FUNCTION_BLOCK "STD_DUMPFlowMonitor"	// FB 1804
TITLE = DUMP-Scale test productflow
//COPYRIGHT:    (C) 2004  BUHLER AG, CH-9240 UZWIL, SWITZERLAND
//
//PRODUCT:      STD_MU664
//
//TITLE:        Test product flow dump scale
//
//              Überprüfen des Produktflusses mit Schüttwaage
//
//
//--------------------------------------------------------------------------------
//
//IDENT:         AUTHOR:             DEPT:                             DATE:
//
//STD_FB1804.3.0 Ph. Engler          MU92                              24-May-2005
//               - InReadyForScaleEmptying
//STD_FB1804.2.0 Ph. Engler          MU92                              11-May-2005
//               - Timer type changed to FB1706
//               - S5Timer 40 changed with an Timer-FB1706
//STD_FB1804.1.0 E.Hanselmann        MU662                             26-Mar-2003
//               1st Release
//
//--------------------------------------------------------------------------------
//
//PURPOSE: 
//
//MANUAL : 
//
//RESTRICTIONS: 
//
//--------------------------------------------------------------------------------
//
AUTHOR : PE
FAMILY : STD
VERSION : 3.0
VAR_INPUT
  InFuncCode : INT ;	//0=nothing,1=DUMP, 2=not used,3=not used,
  InInit : BOOL ;	//(S-DB.ToASW.CmdNewBatch)
  InScaleWeight : DINT ;	//Actual scale weight (#xxx.xxx.OutScaleWeight)
  InJobWeight : DINT ;	//[not used] Actual job weight   (#xxx.xxx.OutJobWeight)
  InFlowrate : DINT ;	//[not used] Actual scale flowrate (#xxx.xxx.OutFlowrate)
  InDumpWeight : INT ;	//Adjusted dump weight scale (#xxx.xxx.DUMP.InDumpWeight)
  InStepScale : INT ;	//Actual scale step  (#xxx.xxx.OutLcStep)
  InFlowMeasureTime : INT ;	//Interval to meassuring product flow (seconds/minutes)
  InMinFlowWeightPerTime : DINT ;	//Minimal weight per messure cycle "NoProductFlow"
  InDelaySeqStopTime : INT ;	//Delay SequenceStop after "NoProductFlow" (seconds/minutes)
  InSectionStarted : BOOL ;	//(S-DB.PcRead.State.StStarted)
  InSectionFeeding : BOOL ;	//(S-DB.PcRead.State.StFeeding)
  InGroupLoaded : BOOL ;	//[not used] (#Gr.OutLoaded)
  InReadyForScaleEmptying : BOOL ;	//The section is ready to monitor the scale for no material flow.
END_VAR
VAR
  FlowMeasureTimer : FB 1706;
  DelaySeqStopTimer : FB 1706;
  WaitForProductDelay : FB 1706;
  OutScaleProductFlowOn : BOOL ;	//Used for "  "
  OutScaleLoaded : BOOL ;	//Used for "  "
  OutReadyRestEmptying : BOOL ;	//Used for cmd "RestEmptying" (#xxx.Ma.InOutEmptyingHopperScale)
  OutProductFlowEnd : BOOL ;	//Used for "SequenzeStop" (S-DB.ToSSW.Func.CmdSequenzStop)
  OutActProductFlowPerTime : DINT ;	//Actual product flow
  ProductWeightOld : DINT ;	//Weight by last cycle
  ProductWeightNew : DINT ;	//Weight by actual cycle
  JobWeightOld : DINT ;	//Weight by last cycle
END_VAR
BEGIN
NETWORK
TITLE = General
      A(;
      L     #InFuncCode;
      L     0;	//Timer type "nothing"
      <=I;
      );
      O;
      A(;
      L     #InFuncCode;
      L     2;	//Timer type "not used"
      >=I;
      );
      BEC;
NETWORK
TITLE = Flow Measure Time Intervall
      NOP   0;
//-Waiting for product---
      L     #InStepScale;
      L     8;	//step wait product
      ==I;
      AN    #FlowMeasureTimer.Q;
      =     #WaitForProductDelay.IN;
// 
      CALL  #WaitForProductDelay (
           TON                      := TRUE,
           ParRestart               := FALSE,
           ParRecalc                := FALSE,
           PT                       := 20);
      L     #InStepScale;
      L     2;
      ==I;
      O     #WaitForProductDelay.Q;
      AN    #FlowMeasureTimer.Q;
// 
//-Intervall for measureing---
      =     #FlowMeasureTimer.IN;
      L     #InFlowMeasureTime;	//step dosing
      T     #FlowMeasureTimer.PT;
//Target Time
      CALL  #FlowMeasureTimer (
           TON                      := TRUE,
           ParRestart               := FALSE,
           ParRecalc                := FALSE);
//Timer
NETWORK
TITLE = Product Flow
      NOP   0;
//Meassure Flow
      L     L#0;
      A     #FlowMeasureTimer.Q;
      JCN   PF04;
      A(;
      L     #InScaleWeight;
      L     L#0;
      <D;
      );
      JC    PF01;
      TAK;
PF01: T     #ProductWeightNew;
// 
      A(;
      L     #ProductWeightNew;
      L     #ProductWeightOld;
      >=D;
      );
      JC    PF02;
      A(;
      L     #ProductWeightNew;
      L     #ProductWeightOld;
      <D;
      );
      JU    PF03;
PF02: L     #ProductWeightNew;
      L     #ProductWeightOld;
      -D;
      JU    PF04;
PF03: L     #InDumpWeight;
      ITD;
      L     1000;	//kg to gr
      *D;
      L     #ProductWeightOld;
      -D;
      L     #ProductWeightNew;
      +D;
      JU    PF04;
PF04: T     #OutActProductFlowPerTime;
      L     #ProductWeightNew;
      T     #ProductWeightOld;
// 
      A(;
      L     #OutActProductFlowPerTime;
      L     #InMinFlowWeightPerTime;
      >=D;
      );
      O(;
      L     #InJobWeight;
      L     #JobWeightOld;
      >D;
      );
      A(;
      O     #InSectionStarted;
      O     #InSectionFeeding;
      );
      S     #OutScaleProductFlowOn;
      S     #OutScaleLoaded;
      A(;
      L     #OutActProductFlowPerTime;
      L     #InMinFlowWeightPerTime;
      <D;
      );
      A     #FlowMeasureTimer.Q;
      R     #OutScaleProductFlowOn;
      L     #InJobWeight;
      T     #JobWeightOld;
// 
//Initialize
      A     #InInit;
      JCN   PF06;
      SET;
      R     #OutScaleProductFlowOn;
      R     #OutScaleLoaded;
      L     L#0;
      T     #ProductWeightNew;
      T     #ProductWeightOld;
      T     #OutActProductFlowPerTime;
PF06: NOP   0;
NETWORK
TITLE = Ready Rest Emptying
      A(;
      O     #InSectionStarted;
      O     #InSectionFeeding;
      );
      A     #FlowMeasureTimer.Q;
      A     #OutScaleLoaded;
      AN    #OutScaleProductFlowOn;
      S     #OutReadyRestEmptying;
//Initialize
      A     #InInit;
      O;
      A     #OutScaleLoaded;
      A     #OutScaleProductFlowOn;
      AN    #InReadyForScaleEmptying;
      R     #OutReadyRestEmptying;
NETWORK
TITLE = Delay SequenzeStop Time
      NOP   0;
//Start
      L     #InDelaySeqStopTime;
      L     0;
      >I;
      A     #InSectionFeeding;
      A     #OutScaleLoaded;
      AN    #OutScaleProductFlowOn;
      =     #DelaySeqStopTimer.IN;
//Target Time
      L     #InDelaySeqStopTime;
      T     #DelaySeqStopTimer.PT;
//Timer
      CALL  #DelaySeqStopTimer (
           TON                      := TRUE,
           ParRestart               := FALSE,
           ParRecalc                := FALSE);
NETWORK
TITLE = Product Flow End
      A     #DelaySeqStopTimer.Q;
      =     #OutProductFlowEnd;
NETWORK
TITLE = End of block
      BE;
END_FUNCTION_BLOCK

FUNCTION_BLOCK "STD_DUMPPulse"	// FB 1805
TITLE = Handling of Scales with Dump Impuls
//COPYRIGHT:    (C) 2004  BUHLER AG, CH-9240 UZWIL, SWITZERLAND
//
//PRODUCT:      STD
//
//TITLE:        Handling of Scales with Dump Impuls
//
//              Schüttimpulsauswertung
//                
// 
//--------------------------------------------------------------------------------
// 
//IDENT:            AUTHOR:             DEPT:                          DATE:
// 
//STD_FB1805.2.0    Ph. Engler          MU664                          03-Jun-2004
//                  Integration to GP-BIB; New functionality
//P02_FB1805.1.1    M.Miotto            MU662                          11-May-2004
//                  Init if no dump after a predefined time >> from 180 decr. 60
//P02_FB1805.1.0    P.Müller            MU662                          30-Apr-2004
//                  1st Release
// 
//--------------------------------------------------------------------------------
// 
//PURPOSE: 
// 
//MANUAL : 
// 
//RESTRICTIONS: 
// 
//--------------------------------------------------------------------------------
//
AUTHOR : PE
FAMILY : STD
VERSION : 2.0
VAR_INPUT
  FunctionCode : INT ;
  InFeeding : BOOL ;
  CmdNewJob : BOOL ;
  CmdNewValue : BOOL ;
  ScalePulse : BOOL ;
  ScalePulseWeight : DINT ;
  TargetFlowrate : INT ;
END_VAR
VAR_OUTPUT
  InfScaleDumpRelease : BOOL ;
END_VAR
VAR_IN_OUT
  ScaleJobWeight : DINT ;
  ScaleNonErasableWeight : DINT ;
  ScaleActualFlowrate : DINT ;
END_VAR
VAR
  TimeCounter : DINT ;
  ScaleDumpTimer : INT ;
  DumpMonitoringTimer : INT ;
  EdgeScalePulse : BOOL ;
  PulseScalePulse : BOOL ;
  ScaleFeeding : BOOL ;
  staFirstDumpDone : BOOL ;
  EdgeInFeeding : BOOL ;
  PulseInFeeding : BOOL ;
  InfDumpMonitoringElapsed : BOOL ;
  staScaleNotDumping : BOOL ;
  staNewFlowrate : BOOL ;
  AverageTime : INT ;
  StartTime : INT ;
  ActDumpIntervallTime : ARRAY  [1 .. 3 ] OF INT ;
END_VAR
VAR_TEMP
  tmpMaxPulsesPerHour : REAL ;
  tmpPulseTime : DINT ;
  tmpNumberOfTimeValues : INT ;
  tmpInputIntervallTime : INT ;
END_VAR
BEGIN
NETWORK
TITLE = Function 1: Calculation of Target Flowrate
      L     #FunctionCode;
      L     1;
      <>I;
      JC    F001;
// 
//-Calculation of Pulse per Hour---
      L     #TargetFlowrate;
      ITD;
      DTR;
      L     #ScalePulseWeight;
      DTR;
      /R;
      T     #tmpMaxPulsesPerHour;
// 
//-Calculation of Pulse Pause---
      L     3.600000e+03;
      L     #tmpMaxPulsesPerHour;
      /R;
      RND;
      T     #tmpPulseTime;
// 
//-Release Scale Dump---
      A     "SYS_Scan0_Tick1s";
      JCN   NE10;
      L     #TimeCounter;
      L     L#1;
      +D;
      T     #TimeCounter;
NE10: L     #tmpPulseTime;
      L     #TimeCounter;
      <=D;
      =     #InfScaleDumpRelease;
      JCN   NE11;
      L     L#0;
      T     #TimeCounter;
NE11: NOP   0;
// 
      BEU;
F001: NOP   0;
NETWORK
TITLE = Function 2: Calculation of Scale Values
//Scale Values:
//- Job Weight
//- Non Erasable Weight
//- Flowrate
      L     #FunctionCode;
      L     2;
      <>I;
      JC    F002;
// 
//-Weight calculatione---
      A     #PulseScalePulse;
      JCN   NE22;
      L     #ScalePulseWeight;
      L     #ScaleJobWeight;
      +D;
      T     #ScaleJobWeight;
// 
      L     #ScalePulseWeight;
      L     #ScaleNonErasableWeight;
      +D;
      T     #ScaleNonErasableWeight;
NE22: NOP   0;
// 
//-Dump intervall time measuring---
      A     #InFeeding;
      A     "SYS_Scan0_Tick1s";
      JCN   NE23;
      L     L#1;
      L     #ScaleDumpTimer;
      +D;
      T     #ScaleDumpTimer;
NE23: NOP   0;
// 
//-CmdNewValue---
      A     #CmdNewValue;
      O     #CmdNewJob;
      S     #staNewFlowrate;
// 
//-Dump monitoring---
      L     0;
//      U     #InFeeding
//      SPBN  DM02
      A     "SYS_Scan0_Tick1s";
      JCN   DM01;
      L     L#1;
      L     #DumpMonitoringTimer;
      +D;
      T     #DumpMonitoringTimer;
DM01: NOP   0;
// 
      AN    #staScaleNotDumping;
      O     #staNewFlowrate;
      JCN   DM03;
      L     #AverageTime;
      L     2;
      /I;
      L     #AverageTime;
      +I;
      JU    DM04;
DM03: L     #AverageTime;
      L     2;
      /I;
DM04: L     #DumpMonitoringTimer;
      <=I;
      A(;
      TAK;
      L     0;
      <>I;
      );
      =     #InfDumpMonitoringElapsed;
      S     #staScaleNotDumping;
// 
//-Number of valid DumpIntervall times---
      L     0;
      T     #tmpNumberOfTimeValues;
      L     #ActDumpIntervallTime[1];
      <>I;
      JCN   AcD1;
      L     1;
      L     #tmpNumberOfTimeValues;
      +I;
      T     #tmpNumberOfTimeValues;
AcD1: L     0;
      L     #ActDumpIntervallTime[2];
      <>I;
      JCN   AcD2;
      L     1;
      L     #tmpNumberOfTimeValues;
      +I;
      T     #tmpNumberOfTimeValues;
AcD2: L     0;
      L     #ActDumpIntervallTime[3];
      <>I;
      JCN   AcD3;
      L     1;
      L     #tmpNumberOfTimeValues;
      +I;
      T     #tmpNumberOfTimeValues;
AcD3: NOP   0;
// 
//-InFeeding---
      A     #InFeeding;
      FP    #EdgeInFeeding;
      =     #PulseInFeeding;
// 
//-Scale dump pulse---
      A     #ScalePulse;
      FP    #EdgeScalePulse;
      =     #PulseScalePulse;
      R     #staScaleNotDumping;
      R     #staNewFlowrate;
// 
//-Save intervall times---
      L     0;
      A     #InfDumpMonitoringElapsed;
      JC    IT01;
      L     #StartTime;
      AN    #staFirstDumpDone;
      JC    IT01;
      L     #ScaleDumpTimer;
IT01: T     #tmpInputIntervallTime;
      A     #PulseScalePulse;
      O     #InfDumpMonitoringElapsed;
      JCN   SI02;
      L     #ActDumpIntervallTime[2];
      T     #ActDumpIntervallTime[3];
      L     #ActDumpIntervallTime[1];
      T     #ActDumpIntervallTime[2];
      L     #tmpInputIntervallTime;
      T     #ActDumpIntervallTime[1];
      L     L#0;
      T     #DumpMonitoringTimer;
      A     #PulseScalePulse;
      JCN   SI02;
      T     #ScaleDumpTimer;
SI02: NOP   0;
// 
//-First dump after inFeeding on---
      A     #PulseScalePulse;
      AN    #staFirstDumpDone;
      S     #staFirstDumpDone;
      AN    #InFeeding;
      R     #staFirstDumpDone;
// 
//-New job/ job change---
      A     #CmdNewJob;
      JCN   NJ01;
//      L     #ActDumpIntervallTime[1]
//      T     #ActDumpIntervallTime[2]
//      L     0
//      T     #ActDumpIntervallTime[1]
//      T     #ActDumpIntervallTime[3]
// 
      L     L#0;
      T     #ScaleJobWeight;
NJ01: NOP   0;
// 
//-Time average---
      L     #ActDumpIntervallTime[1];
      L     #ActDumpIntervallTime[2];
      +I;
      L     #ActDumpIntervallTime[3];
      +I;
      L     #tmpNumberOfTimeValues;
      /I;
      T     #AverageTime;
// 
//-Start time---
      L     0;
      L     #AverageTime;
      <>I;
      JCN   ST01;
      L     #AverageTime;
      T     #StartTime;
ST01: NOP   0;
// 
//-Flowrate---
      L     0;
      A     #InFeeding;
      JCN   FL01;
      L     #ScalePulseWeight;
      L     L#3600;
      *D;
      L     #AverageTime;
      /D;
FL01: T     #ScaleActualFlowrate;
// 
//-Scale feeding---
      L     #ScaleActualFlowrate;
      L     0;
      >I;
      A     #InFeeding;
      =     #ScaleFeeding;
// 
      SET;
      R     #CmdNewValue;
      R     #CmdNewJob;
// 
      BEU;
F002: NOP   0;
NETWORK
TITLE = End of block
      BE;
END_FUNCTION_BLOCK

// FC 6: know-how protected block, not included

// FC 8: know-how protected block, not included

FUNCTION "SYS_DPDiag1" : VOID	// FC 76
TITLE = DP-additional Diag
//COPYRIGHT:     (C) 2001 BY  BUEHLER LTD. 
//                            CH-9240 UZWIL  SWITZERLAND
//
//PRODUCT:       DP-Diagnosis
//
//TITLE:         DP-additional Diag
//
//-------------------------------------------------------------------------
//
//IDENT:        AUTOR:              DEPT:                         DATE:
//
//FC76.2.0      Ph. Engler          MU664                        14-Dec-2004
//              Wago 750-333: Corrections and adaption to WinCC
//FC76.1B       K. Tischer          CT3                          20-Feb-2003
//              new buskoppler Wago 750-333 added
//FC76.1A       K. Tischer          CT3                          28-MAY-2001
//              1st Release
//
//-------------------------------------------------------------------------
//
//PURPOSE:  - each mastersystem is a separate Network
//              - initial same Bit
//              - Call DP-Diagnostic (orig. Siemens) 
//              - Call additional Diagnostic for not Siemens Slaves
//              - reset same parameters
//
//RESTRICTIONS:   NEEDS SIEMENS FB76 (original FB125)
//                NEEDS FC75 Main Diagnostic
//
//
//-------------------------------------------------------------------------
//
//
AUTHOR : PE
FAMILY : DP
NAME : DPDiag1
VERSION : 2.0
VAR_TEMP
  Sum_Slave_Diag_Int : BYTE ;	//summary Slave Diagnosen
  ErrorNo : BYTE ;	//TiK
  ByteStart : INT ;	//TiK
  Diag_Lentgh : BYTE ;	//TiK
  Adr : DINT ;	//adress1
  Adr2 : DINT ;	//Adress 2
END_VAR
BEGIN
NETWORK
TITLE = check is diagtic present
      AN    DBX 932.3;	// additional diagnostic data present
      BEC;
NETWORK
TITLE = WAxx Wago (B750) 
//additianal Diagnisis for Wago Slaves Type (B750)
//
// - check result from SIEMENS FB76 => error type = device diagnosis
// - check result from SIEMENS FB76 => slave ident = B750
//
      NOP   0;
// error type = device diagnosis
      A(;
      L     DBB 11;	// error typ
      L     5;	// check device diagnostic
      ==I;
      );
// slave ident = B750
      A(;
      L     DBW 8;	// slave ident
      L     W#16#B750;	// B750 = Wago
      ==I;
      );
      JCN   WA00;	// jump end
// Init wago standard
      L     8;	// standard length of wago diagnostic data
      T     #Diag_Lentgh;
      L     DBB 1398;	// old error no (stored)
      T     #ErrorNo;	// error no
// calc summary DiagData
      L     DBB 938;	// norm diag data byte 6 (length)
      +     -2;	// 2 byte length info
      L     #Diag_Lentgh;	// Wago standard length =8
      /I;
      T     #Sum_Slave_Diag_Int;	// summary diag data
// Diag counter intialisieren
      A     DBX 2.3;	// single step error
      JCN   WA07;
// Diag counter inkrementieren
      L     #ErrorNo;	// actual diagnostic data no
      +     1;	// inkrement 1
      T     #ErrorNo;	// actual diagnostic data no
// Diag conter upper and lower limit
WA07: A(;
      L     #ErrorNo;
      L     #Sum_Slave_Diag_Int;	// upper limit 
      >I;
      );
      O(;
      L     #ErrorNo;
      L     1;	// lower limit
      <I;
      );
      JCN   WA06;
      L     1;	// set count diag =1
      T     #ErrorNo;	// out of range
WA06: NOP   0;
// write diagnostic to siemens DB
      L     #ErrorNo;
      T     DBB 10;	// => error number
      T     DBB 1398;	// => reserve byte siemens to store old error number
// calc start byte
      L     #ErrorNo;	// actual diagnostic data no
      L     #Diag_Lentgh;	// length diagnostic data
      *D;	// offset to start byte
      L     932;	// start byte diagnostic data
      +D;
      T     #ByteStart;	// => byte src diagnostic data
// ==check for Profibus or Klemmbus Diagnosis (first byte diagnostic data=0)===================      
      L     0;	// byte no
      L     #ByteStart;	// byte no start actual data
      +D;
      SLD   3;	// convert to bit value
      T     #Adr;	// store bit value
      L     DBB [#Adr];	// first byte diagnostic data
      L     0;
      ==I;
      JC    WA02;	//>>jump to check Klembus diagnosis >>>>>>>>>>>>>>>>>>>
// Modul / Kanal Diagnose ============================
      L     DBB [#Adr];	// first byte diagnostic data
      T     DBB 12;	// => modul no
      L     1;	// byte no
      L     #ByteStart;	// byte no start actual data
      +D;
      SLD   3;	// convert to bit value
      T     #Adr;	// store bit value
      L     DBB [#Adr];
      T     DBB 14;	// => cannel no
// Error analyse
      L     4;	// byte no
      L     #ByteStart;	// byte no start actual data
      +D;
      SLD   3;	// convert to bit value
      T     #Adr;	// store bit value
// == check Lower limit violated ======
      L     DBB [#Adr];
      L     2#100000001;	// compare bit 0 set
      AW;
      L     0;
      JCN   WA05;	// >> jump to check overrange >>>>>>>>>>>>>>>>>>>>>>>>>
      L     8;	//  8=Lower limit violated
      JU    WA03;	// >> jump to => canal error code >>>>>>>>>>>>>>>>>>>>>
// == check Upper limit violated ======
WA05: L     DBB [#Adr];
      L     2#100000010;	// compare bit 1 set
      AW;
      JCN   WA04;	// >> jump to other fault
      L     7;	// 7=Upper limit violated
      JU    WA03;	// >> jump to => canal error code >>>>>>>>>>>>>>>>>>>>>
WA04: L     DBB [#Adr];
      L     2#101000000;	// compare bit 6 set
      AW;
      JCN   WA03;	// >> jump to => canal error code >>>>>>>>>>>>>>>>>>>>>
      L     9;	// 9= Fault (e.g. encoder supply, load voltage at the output...;
WA03: T     DBW 16;	// => canal error code
      L     3;	// 3= channel error
      T     DBB 11;	// => error type
      JU    WA00;	// jump end
WA02: NOP   0;	// << check Klemmbus diagnosis <<<<<<<<<<<<<<<<<<<<<<<<<
      L     1;	// byte no
      L     #ByteStart;	// byte no start actual data
      +D;
      SLD   3;	// convert to bit value
      T     #Adr;	// store bit value
      L     DBB [#Adr];
      L     0;
      ==I;
      JC    WA01;	//>>jump to Klemmbus diagnosis >>>>>>>>>>>>>>>>>>>>>>>>>
// Profibus Diagnosis =================================
      L     4;	// byte no
      L     #ByteStart;	// byte no start actual data
      +D;
      SLD   3;	// convert to bit value
      T     #Adr;	// store bit value
      L     DBB [#Adr];
      L     100;	// 100=not enough configuration data;200=error in 1st configuration byte;300=non-supported module at position N
      *I;
      T     DBB 13;	// => modul state
      L     2;	// 2=Modul Diagnosis
      T     DBB 11;	// => error type
      JU    WA00;	// >> jump end >>>>>>>>>>>>>>>>>>>>>>>>>>>>>>>>>>>>>>>>>>>
// << Klemmenbus Diagnosis <<<<<<<<<<<<<<<<<<<<<<<<<<<<<<<
WA01: NOP   0;
// prepair modul no
      L     5;	// byte no
      L     #ByteStart;	// byte no start actual data
      +D;
      SLD   3;	// convert to bit value
      T     #Adr;	// store bit value
      L     DBB [#Adr];
      T     DBB 12;	// => modul no
// prepair modul state
      L     4;	// byte no
      L     #ByteStart;	// byte no start actual data
      +D;
      SLD   3;	// convert to bit value
      T     #Adr;	// store bit value
      L     DBB [#Adr];
      L     10;	// 10=EEPROM Checksum Error;20=error in programmed process image;30=modules have identified error in fieldbus commands;40=fieldbus break after module N
      *I;	// 50=filedbus error in register communication with module N;60=error in PROFIBUS-DP configuration telegram;70=non-supported module at position N
      T     DBB 13;	// => modul state
// prepair error type
      L     2;	// 2=Modul Diagnosis
      T     DBB 11;	// => error type
      JU    WA00;	// jump end
WA00: NOP   0;
NETWORK
TITLE = WAxx Wago (B754) 
//additianal Diagnisis for Wago Slaves Type (B750-333)
//
// - check result from SIEMENS FB76 => error type = device diagnosis
// - check result from SIEMENS FB76 => slave ident = B750
//
      NOP   0;
// error type = device diagnosis
      A(;
      L     DBB 11;	// error typ
      L     5;	// check device diagnostic
      ==I;
      );
// slave ident = B750-333
      A(;
      L     DBW 8;	// slave ident
      L     W#16#B754;	// B754 = Wago
      ==I;
      );
      JCN   WB00;	// jump end
// Init wago standard
      L     3;
      T     #Diag_Lentgh;	// kanaldiagsostic standard length =3
      L     DBB 1398;	// old error no (stored)
      T     #ErrorNo;	// error no
// calc summary DiagData
      L     DBB 44;	// length of diagnostic data (SFC13) incl. header
      L     22;	// 22 byte (header=6Byte; kennungdata=9Byte; modulstate=7
      >=I;
      JCN   WB00;
      L     DBB 44;	// length of diagnostic data (SFC13) incl. header
      +     -22;	// 22 byte (header=6Byte; kennungdata=9Byte; modulstate=7
      L     3;	// Wago standard length =3
      /I;
      T     #Sum_Slave_Diag_Int;	// summary diag data
// Diag counter intialisieren
      A     DBX 2.3;	// single step error
      JCN   WB07;
// Diag counter inkrementieren
      L     #ErrorNo;	// actual diagnostic data no
      +     1;	// inkrement 1
      T     #ErrorNo;	// actual diagnostic data no
// Diag conter upper and lower limit
WB07: A(;
      L     #ErrorNo;
      L     #Sum_Slave_Diag_Int;	// upper limit 
      >I;
      );
      O(;
      L     #ErrorNo;
      L     1;	// lower limit
      <I;
      );
      JCN   WB06;
      L     1;	// set error no =1
      T     #ErrorNo;	// out of range
WB06: NOP   0;
// write diagnostic to siemens DB
      L     #ErrorNo;
      T     DBB 10;	// => error number
      T     DBB 1398;	// => reserve byte siemens to store old error number
// ==check for Profibus or Klemmbus Diagnosis (first byte diagnostic data=0)===================      
      L     951;	//byte 20 => device diagnostic 
      SLD   3;
      T     #Adr;
      L     952;
      SLD   3;
      T     #Adr2;
      L     DBB [#Adr];	// state message 0= no error
      L     0;
      >I;
      JCN   WB10;
      L     2;	// 2=Modul Diagnosis
      T     DBB 11;	// => error type
//-PE-Begin---
      L     DBB [#Adr];
      L     W#16#1;
      ==I;
      JCN   PE01;
      L     10;
      L     DBB [#Adr2];
      +I;
      JU    PESA;
// 
PE01: L     DBB [#Adr];
      L     W#16#2;
      ==I;
      JCN   PE02;
      L     21;
      L     DBB [#Adr2];
      +I;
      JU    PESA;
// 
PE02: L     DBB [#Adr];
      L     W#16#44;
      ==I;
      A(;
      L     DBB [#Adr2];
      L     0;
      ==I;
      );
      JCN   PE03;
      L     90;
      JU    PESA;
// 
PE03: L     DBB [#Adr];
      L     W#16#81;
      ==I;
      A(;
      L     DBB [#Adr2];
      L     W#16#1;
      ==I;
      );
      JCN   PE04;
      L     91;
      JU    PESA;
// 
PE04: L     DBB [#Adr];
      L     W#16#81;
      ==I;
      A(;
      L     DBB [#Adr2];
      L     W#16#2;
      ==I;
      );
      JCN   PE05;
      L     92;
      JU    PESA;
// 
PE05: L     DBB [#Adr];
      L     W#16#83;
      ==I;
      A(;
      L     DBB [#Adr2];
      L     W#16#1;
      ==I;
      );
      JCN   PE06;
      L     93;
      JU    PESA;
// 
PE06: L     DBB [#Adr];
      L     W#16#83;
      ==I;
      A(;
      L     DBB [#Adr2];
      L     W#16#2;
      ==I;
      );
      JCN   PE07;
      L     94;
      JU    PESA;
// 
PE07: L     DBB [#Adr];
      L     W#16#85;
      ==I;
      A(;
      L     DBB [#Adr2];
      L     W#16#1;
      ==I;
      );
      JCN   PE08;
      L     95;
      JU    PESA;
// 
PE08: L     DBB [#Adr];
      L     W#16#85;
      ==I;
      A(;
      L     DBB [#Adr2];
      L     W#16#2;
      ==I;
      );
      JCN   PE09;
      L     96;
      JU    PESA;
// 
PE09: L     DBB [#Adr];
      L     W#16#86;
      ==I;
      A(;
      L     DBB [#Adr2];
      L     W#16#1;
      ==I;
      );
      JCN   PE10;
      L     97;
      JU    PESA;
// 
PE10: L     DBB [#Adr];
      L     W#16#86;
      ==I;
      A(;
      L     DBB [#Adr2];
      L     W#16#2;
      ==I;
      );
      JCN   PE98;
      L     98;
      JU    PESA;
PESA: T     DBB 13;	// => modul state
      JU    PE99;
PE98: NOP   0;
      L     DBB [#Adr];
      T     DBB 13;	// => modul state
PE99: NOP   0;
//-PE-End---
      L     DBB [#Adr2];
      T     DBB 12;	// => modul no
      L     0;
      T     DBW 16;	// => error no
      JU    WB00;	// >> jump end >>>>>>>>>>>>>>>>>>>>>>>>>>>>>>>>>>>>>>>>>>>
// << Klemmenbus Diagnosis <<<<<<<<<<<<<<<<<<<<<<<<<<<<<<<
WB10: NOP   0;
// calc start byte
      L     #ErrorNo;	// actual diagnostic data no
      L     #Diag_Lentgh;	// length diagnostic data (3Byte)
      *D;	// offset to start byte
      L     951;	// start byte diagnostic data
      +D;
      T     #ByteStart;	// => byte src diagnostic data
// Kanal Diagnose ============================
      L     3;	// 3= channel error
      T     DBB 11;	// => error type
      L     #ByteStart;
      SLD   3;
      T     #Adr;
      L     DBB [#Adr];	// first byte diagnostic data
      L     B#16#3F;
      AW;
      T     DBB 12;	// => modul no
      L     1;	// byte no
      L     #ByteStart;	// byte no start actual data
      +D;
      SLD   3;	// convert to bit value
      T     #Adr;	// store bit value
      L     DBB [#Adr];
      L     B#16#3F;
      AW;
      T     DBB 14;	// => cannel no
      L     2;	// byte no
      L     #ByteStart;	// byte no start actual data
      +D;
      SLD   3;	// convert to bit value
      T     #Adr;	// store bit value
      L     DBB [#Adr];
      L     B#16#1F;
      AW;
      L     600;	//PE
      +I;	//PE
      T     DBW 16;	// => error no
WB00: NOP   0;
END_FUNCTION

FUNCTION "ASW_GraphicFunction" : VOID	// FC 80
TITLE = Display animation; Graphic display data, function keys
//COPYRIGHT:    (C) 2003 BY  BUHLER AG
//                           CH-9240 UZWIL  SWITZERLAND
//
//PRODUCT:      YYY_YYYxx_xx
//
//TITLE:        Prepare Data for Visualisation Interface in DB80
//
//              Aufbereitung der Visualisierungsdaten im DB80
//              
//
//--------------------------------------------------------------------------------
//
//IDENT:        AUTHOR:             DEPT:                               DATE:
//
//P01_FC080.1A  CH. Ebneter         FU53                                4-Mar-2003
//              1st Release
//
//--------------------------------------------------------------------------------
//
//PURPOSE:      
//
//RESTRICTIONS: 
//
//-------------------------------------------------------------------------
//
AUTHOR : CE
FAMILY : USW
VERSION : 0.0
VAR_TEMP
  tmpStartNext : BOOL ;	//Condition to Start next element
  tmpFlagFault : BOOL ;	//Flag mechanical fault
  tmpEnableFeed : BOOL ;
  tmpSndBin : INT ;
  tmpRcvBin : INT ;
END_VAR
BEGIN
NETWORK
TITLE = Global
      A     M 50.0;
      BEU;
//-> Implement for each line a segment
//-> Make all data transfer into the DB80
      =     M 50.0;
      NOP   0;
//-Raw wheat bin discharges---
      L     0;
      T     "ASW_GraphicData".GraficDisplayData.Value1;
      L     0;
      T     "ASW_GraphicData".GraficDisplayData.Value2;
      L     0;
      T     "ASW_GraphicData".GraficDisplayData.Value3;
NETWORK
TITLE = L01INT1 Intake and turnover
      NOP   0;
//-Actual job weight---
      L     0;
      T     "ASW_GraphicData".GraficDisplayData.Value4;
NETWORK
TITLE = If you implement a MU-plant, please delete all further segments
NETWORK
TITLE = Horn quitt from visualisation
// Set CmdHornOff in each line
      A     "ASW_GraphicData".General.Horn.Quit[1];
//      S     "L01".ToSSW.Func.CmdHornOff
      R     "ASW_GraphicData".General.Horn.Quit[1];
NETWORK
TITLE = Reset Emergency stop system from visualisation
      A     "ASW_GraphicData".General.EmergencyStop.SystemReset;
      R     "ASW_GraphicData".General.EmergencyStop.SystemReset;
NETWORK
TITLE = Animation function key SF01
//      O(                                     // Example
//      O     "L11S01".Fault.EsBatchSize
//      O     "L11S01".Fault.EsRefillLevel
//      O     "L11S01".Fault.EsSectionTimeOut
//      O     "L11S01".Fault.EsHandAddTimeOut
//      O     "L11S01".Fault.EsRecipePlace
//      O     "L11S01".Fault.EsProductMismatch
//      O     "L11S01".Fault.Es22
//      O     "L11S01".Fault.Es23
//      O     "L11S01".Fault.EsEmpty
//      O     "L11S01".Fault.ESFull
//      O     "L11S01".Fault.EsWayConflict
//      O     "L11S01".Fault.EsWarning
//      O     "L11S01".Fault.EsMech
//      O     "L11S01".Fault.EsDosing
//      U     "L11S01".ToASW.InfDataReady
//      )     
      =     "ASW_GraphicData".Buttons.Fault_SF.F1;
//      O     "L11S01".Status.StaHand       // Example
      AN    "ASW_GraphicData".Buttons.Fault_SF.F1;
      =     "ASW_GraphicData".Buttons.Manual_SF.F1;
//      O     "L11S01".ToASW.InfDataReady    // Example
      AN    "ASW_GraphicData".Buttons.Fault_SF.F1;
      AN    "ASW_GraphicData".Buttons.Manual_SF.F1;
      =     "ASW_GraphicData".Buttons.Active_SF.F1;
NETWORK
TITLE = Animation function key SF02
      CLR;
      =     "ASW_GraphicData".Buttons.Fault_SF.F2;
      CLR;
      AN    "ASW_GraphicData".Buttons.Fault_SF.F2;
      =     "ASW_GraphicData".Buttons.Manual_SF.F2;
      CLR;
      AN    "ASW_GraphicData".Buttons.Fault_SF.F2;
      AN    "ASW_GraphicData".Buttons.Manual_SF.F2;
      =     "ASW_GraphicData".Buttons.Active_SF.F2;
NETWORK
TITLE = Animation function key SF03
      CLR;
      =     "ASW_GraphicData".Buttons.Fault_SF.F3;
      CLR;
      AN    "ASW_GraphicData".Buttons.Fault_SF.F3;
      =     "ASW_GraphicData".Buttons.Manual_SF.F3;
      CLR;
      AN    "ASW_GraphicData".Buttons.Fault_SF.F3;
      AN    "ASW_GraphicData".Buttons.Manual_SF.F3;
      =     "ASW_GraphicData".Buttons.Active_SF.F3;
NETWORK
TITLE = Animation function key SF04
      CLR;
      =     "ASW_GraphicData".Buttons.Fault_SF.F4;
      CLR;
      AN    "ASW_GraphicData".Buttons.Fault_SF.F4;
      =     "ASW_GraphicData".Buttons.Manual_SF.F4;
      CLR;
      AN    "ASW_GraphicData".Buttons.Fault_SF.F4;
      AN    "ASW_GraphicData".Buttons.Manual_SF.F4;
      =     "ASW_GraphicData".Buttons.Active_SF.F4;
NETWORK
TITLE = Animation function key SF05
      CLR;
      =     "ASW_GraphicData".Buttons.Fault_SF.F5;
      CLR;
      AN    "ASW_GraphicData".Buttons.Fault_SF.F5;
      =     "ASW_GraphicData".Buttons.Manual_SF.F5;
      CLR;
      AN    "ASW_GraphicData".Buttons.Fault_SF.F5;
      AN    "ASW_GraphicData".Buttons.Manual_SF.F5;
      =     "ASW_GraphicData".Buttons.Active_SF.F5;
NETWORK
TITLE = Animation function key SF06
      CLR;
      =     "ASW_GraphicData".Buttons.Fault_SF.F6;
      CLR;
      AN    "ASW_GraphicData".Buttons.Fault_SF.F6;
      =     "ASW_GraphicData".Buttons.Manual_SF.F6;
      CLR;
      AN    "ASW_GraphicData".Buttons.Fault_SF.F6;
      AN    "ASW_GraphicData".Buttons.Manual_SF.F6;
      =     "ASW_GraphicData".Buttons.Active_SF.F6;
NETWORK
TITLE = Animation function key SF07
      CLR;
      =     "ASW_GraphicData".Buttons.Fault_SF.F7;
      CLR;
      AN    "ASW_GraphicData".Buttons.Fault_SF.F7;
      =     "ASW_GraphicData".Buttons.Manual_SF.F7;
      CLR;
      AN    "ASW_GraphicData".Buttons.Fault_SF.F7;
      AN    "ASW_GraphicData".Buttons.Manual_SF.F7;
      =     "ASW_GraphicData".Buttons.Active_SF.F7;
NETWORK
TITLE = Animation function key SF08
      CLR;
      =     "ASW_GraphicData".Buttons.Fault_SF.F8;
      CLR;
      AN    "ASW_GraphicData".Buttons.Fault_SF.F8;
      =     "ASW_GraphicData".Buttons.Manual_SF.F8;
      CLR;
      AN    "ASW_GraphicData".Buttons.Fault_SF.F8;
      AN    "ASW_GraphicData".Buttons.Manual_SF.F8;
      =     "ASW_GraphicData".Buttons.Active_SF.F8;
NETWORK
TITLE = Animation function key SF09
      CLR;
      =     "ASW_GraphicData".Buttons.Fault_SF.F9;
      CLR;
      AN    "ASW_GraphicData".Buttons.Fault_SF.F9;
      =     "ASW_GraphicData".Buttons.Manual_SF.F9;
      CLR;
      AN    "ASW_GraphicData".Buttons.Fault_SF.F9;
      AN    "ASW_GraphicData".Buttons.Manual_SF.F9;
      =     "ASW_GraphicData".Buttons.Active_SF.F9;
NETWORK
TITLE = Animation function key SF10
      CLR;
      =     "ASW_GraphicData".Buttons.Fault_SF.F10;
      CLR;
      AN    "ASW_GraphicData".Buttons.Fault_SF.F10;
      =     "ASW_GraphicData".Buttons.Manual_SF.F10;
      CLR;
      AN    "ASW_GraphicData".Buttons.Fault_SF.F10;
      AN    "ASW_GraphicData".Buttons.Manual_SF.F10;
      =     "ASW_GraphicData".Buttons.Active_SF.F10;
NETWORK
TITLE = Animation function key F1
      CLR;
      =     "ASW_GraphicData".Buttons.Fault_F.F1;
      CLR;
      AN    "ASW_GraphicData".Buttons.Fault_F.F1;
      =     "ASW_GraphicData".Buttons.Manual_F.F1;
      CLR;
      AN    "ASW_GraphicData".Buttons.Fault_F.F1;
      AN    "ASW_GraphicData".Buttons.Manual_F.F1;
      =     "ASW_GraphicData".Buttons.Active_F.F1;
NETWORK
TITLE = Animation function key F02
      CLR;
      =     "ASW_GraphicData".Buttons.Fault_F.F2;
      CLR;
      AN    "ASW_GraphicData".Buttons.Fault_F.F2;
      =     "ASW_GraphicData".Buttons.Manual_F.F2;
      CLR;
      AN    "ASW_GraphicData".Buttons.Fault_F.F2;
      AN    "ASW_GraphicData".Buttons.Manual_F.F2;
      =     "ASW_GraphicData".Buttons.Active_F.F2;
NETWORK
TITLE = Animation function key F03
      CLR;
      =     "ASW_GraphicData".Buttons.Fault_F.F3;
      CLR;
      AN    "ASW_GraphicData".Buttons.Fault_F.F3;
      =     "ASW_GraphicData".Buttons.Manual_F.F3;
      CLR;
      AN    "ASW_GraphicData".Buttons.Fault_F.F3;
      AN    "ASW_GraphicData".Buttons.Manual_F.F3;
      =     "ASW_GraphicData".Buttons.Active_F.F3;
NETWORK
TITLE = Animation function key F04
      CLR;
      =     "ASW_GraphicData".Buttons.Fault_F.F4;
      CLR;
      AN    "ASW_GraphicData".Buttons.Fault_F.F4;
      =     "ASW_GraphicData".Buttons.Manual_F.F4;
      CLR;
      AN    "ASW_GraphicData".Buttons.Fault_F.F4;
      AN    "ASW_GraphicData".Buttons.Manual_F.F4;
      =     "ASW_GraphicData".Buttons.Active_F.F4;
NETWORK
TITLE = Animation function key F05
      CLR;
      =     "ASW_GraphicData".Buttons.Fault_F.F5;
      CLR;
      AN    "ASW_GraphicData".Buttons.Fault_F.F5;
      =     "ASW_GraphicData".Buttons.Manual_F.F5;
      CLR;
      AN    "ASW_GraphicData".Buttons.Fault_F.F5;
      AN    "ASW_GraphicData".Buttons.Manual_F.F5;
      =     "ASW_GraphicData".Buttons.Active_F.F5;
NETWORK
TITLE = Animation function key F06
      CLR;
      =     "ASW_GraphicData".Buttons.Fault_F.F6;
      CLR;
      AN    "ASW_GraphicData".Buttons.Fault_F.F6;
      =     "ASW_GraphicData".Buttons.Manual_F.F6;
      CLR;
      AN    "ASW_GraphicData".Buttons.Fault_F.F6;
      AN    "ASW_GraphicData".Buttons.Manual_F.F6;
      =     "ASW_GraphicData".Buttons.Active_F.F6;
NETWORK
TITLE = Animation function key F07
      CLR;
      =     "ASW_GraphicData".Buttons.Fault_F.F7;
      CLR;
      AN    "ASW_GraphicData".Buttons.Fault_F.F7;
      =     "ASW_GraphicData".Buttons.Manual_F.F7;
      CLR;
      AN    "ASW_GraphicData".Buttons.Fault_F.F7;
      AN    "ASW_GraphicData".Buttons.Manual_F.F7;
      =     "ASW_GraphicData".Buttons.Active_F.F7;
NETWORK
TITLE = Animation function key F08
      CLR;
      =     "ASW_GraphicData".Buttons.Fault_F.F8;
      CLR;
      AN    "ASW_GraphicData".Buttons.Fault_F.F8;
      =     "ASW_GraphicData".Buttons.Manual_F.F8;
      CLR;
      AN    "ASW_GraphicData".Buttons.Fault_F.F8;
      AN    "ASW_GraphicData".Buttons.Manual_F.F8;
      =     "ASW_GraphicData".Buttons.Active_F.F8;
NETWORK
TITLE = Animation function key F09
      CLR;
      =     "ASW_GraphicData".Buttons.Fault_F.F9;
      CLR;
      AN    "ASW_GraphicData".Buttons.Fault_F.F9;
      =     "ASW_GraphicData".Buttons.Manual_F.F9;
      CLR;
      AN    "ASW_GraphicData".Buttons.Fault_F.F9;
      AN    "ASW_GraphicData".Buttons.Manual_F.F9;
      =     "ASW_GraphicData".Buttons.Active_F.F9;
NETWORK
TITLE = Animation function key F10
      CLR;
      =     "ASW_GraphicData".Buttons.Fault_F.F10;
      CLR;
      AN    "ASW_GraphicData".Buttons.Fault_F.F10;
      =     "ASW_GraphicData".Buttons.Manual_F.F10;
      CLR;
      AN    "ASW_GraphicData".Buttons.Fault_F.F10;
      AN    "ASW_GraphicData".Buttons.Manual_F.F10;
      =     "ASW_GraphicData".Buttons.Active_F.F10;
NETWORK
TITLE = Way animation picture F01
      CLR;
      =     "ASW_GraphicData".Way.F01.L0.B0;
NETWORK
TITLE = Way animation picture F02
      CLR;
      =     "ASW_GraphicData".Way.F02.L0.B0;
NETWORK
TITLE = Way animation picture F03
      CLR;
      =     "ASW_GraphicData".Way.F03.L0.B0;
NETWORK
TITLE = Way animation picture F04
      CLR;
      =     "ASW_GraphicData".Way.F04.L0.B0;
NETWORK
TITLE = Way animation picture F05
      CLR;
      =     "ASW_GraphicData".Way.F05.L0.B0;
NETWORK
TITLE = Way animation picture F06
      CLR;
      =     "ASW_GraphicData".Way.F06.L0.B0;
NETWORK
TITLE = Way animation picture F07
      CLR;
      =     "ASW_GraphicData".Way.F07.L0.B0;
NETWORK
TITLE = Way animation picture F08
      CLR;
      =     "ASW_GraphicData".Way.F08.L0.B0;
NETWORK
TITLE = Way animation picture F09
      CLR;
      =     "ASW_GraphicData".Way.F09.L0.B0;
NETWORK
TITLE = Way animation picture F10
      CLR;
      =     "ASW_GraphicData".Way.F10.L0.B0;
NETWORK
TITLE = Way animation picture SF01
      CLR;
      =     "ASW_GraphicData".Way.SF01.L0.B0;
NETWORK
TITLE = Way animation picture SF02
      CLR;
      =     "ASW_GraphicData".Way.SF02.L0.B0;
NETWORK
TITLE = Way animation picture SF03
      CLR;
      =     "ASW_GraphicData".Way.SF03.L0.B0;
NETWORK
TITLE = Way animation picture SF04
      CLR;
      =     "ASW_GraphicData".Way.SF04.L0.B0;
NETWORK
TITLE = Way animation picture SF05
      CLR;
      =     "ASW_GraphicData".Way.SF05.L0.B0;
NETWORK
TITLE = Way animation picture SF06
      CLR;
      =     "ASW_GraphicData".Way.SF06.L0.B0;
NETWORK
TITLE = Way animation picture SF07
      CLR;
      =     "ASW_GraphicData".Way.SF07.L0.B0;
NETWORK
TITLE = Way animation picture SF08
      CLR;
      =     "ASW_GraphicData".Way.SF08.L0.B0;
NETWORK
TITLE = Way animation picture SF09
      CLR;
      =     "ASW_GraphicData".Way.SF09.L0.B0;
NETWORK
TITLE = Way animation picture SF10
      CLR;
      =     "ASW_GraphicData".Way.SF10.L0.B0;
END_FUNCTION

FUNCTION "ASW_PlantParFunction" : VOID	// FC 81
TITLE = Plant parameters and date/time setting
//
//COPYRIGHT:      (C) 2000 BY  BUHLER LTD.
//                           CH-9240 UZWIL  SWITZERLAND
//
//PRODUCT:        GEN_MU664
//
//TITLE:          Plant parameters and date/time setting
//
//                Anlagen parameter und Datum/Uhrzeit-Einstellung
//
//
//--------------------------------------------------------------------------------
//
//IDENT:          AUTOR:            DEPT:                              DATE:
//
//GEN_FC081.3.0   Ph. Engler        MU664                              27-Feb-2004
//                - Plant specific commands and parameters deleted
//GEN_FC081.2.0   Ph. Engler        MU664                              06-Jan-2004
//                - Time setting changed: Seconds instead of Milliseconds
//GEN_FC081.1.0   Ph. Engler        MU664                              05-Mar-2003
//                1st Release
//
//--------------------------------------------------------------------------------
//
//PURPOSE:      
//
//RESTRICTIONS: 
//
//--------------------------------------------------------------------------------
//
//
AUTHOR : CE
FAMILY : GEN
VERSION : 0.0
VAR_TEMP
  tmpDateTime : DATE_AND_TIME ;
  tmpPafe : INT ;
  tmpDATE : DATE ;
  tmpTOD : TIME_OF_DAY ;
  tmpBool : BOOL ;
  tmpDWORD : DWORD ;
END_VAR
BEGIN
NETWORK
TITLE = DT Copy date and time from PCS to PLC
      L     DB81.DBW 10;
      L     0;
      ==I;
      JC    DT00;
// 
//-Create Any-Pointer---
      L     DB81.DBW 10;
      T     #tmpDATE;
      L     DB81.DBW 12;
      L     L#60000;
      *D;
      T     #tmpTOD;
      L     DB81.DBW 14;
      L     L#1000;
      *D;
      L     #tmpTOD;
      +D;
      T     #tmpTOD;
// 
      CALL  "SIEMENS.IECFC3.TOD_DT" (
           $1                       := #tmpDATE,
           $2                       := #tmpTOD,
           $3                       := #tmpDateTime);
// 
// Set CPU time
      CALL  SFC 0 (
           PDT                      := #tmpDateTime,
           RET_VAL                  := #tmpPafe);
// 
// reset Data from PCS
      L     0;
      T     DB81.DBW 10;
      T     DB81.DBW 12;
      T     DB81.DBW 14;
DT00: NOP   0;
NETWORK
TITLE = End of block
      BE;
END_FUNCTION

// FC 92: know-how protected block, not included

FUNCTION "SYS_GeneralPLCStartup" : VOID	// FC 100
TITLE = General plc startup functions
//COPYRIGHT:      (C) 2000 BY  BUHLER LTD.
//                           CH-9240 UZWIL  SWITZERLAND
//
//PRODUCT:        MELE_SMU01_99
//
//TITLE:          General PLC startup functions
//
//                Generelle SPS-Anlauffunktionen
//
//
//--------------------------------------------------------------------------------
//
//IDENT:          AUTOR:            DEPT:                              DATE:
//
//P0x_FC100.3.2   Ph. Engler        MU664                              27-Jul-2005
//                Simulation initalized
//P0x_FC100.3.1   Ph. Engler        MU664                              15-Nov-2004
//                Set all HW-Stop-Flags
//P0x_FC100.3.0   Ph. Engler        MU664                              07-Feb-2003
//                Redesign GCS7 Release 2
//P0x_FC100.2.1   Ph. Engler        MU664                              26-Oct-2002
//                Command CmdStartTestMode integrated
//P0x_FC100.2.0   Ph. Engler        MU664                              21-Dec-2000
//                ColdStart for CPU 416-2 implemented
//                (requires DB50.1.1 or higher)
//P01_FC100.1.0   Ph. Engler        MU664                              05-Jan-2000
//                1st Release
//
//--------------------------------------------------------------------------------
//
//PURPOSE:      
//
//RESTRICTIONS: 
//
//--------------------------------------------------------------------------------
//
//
AUTHOR : PE
FAMILY : USW
VERSION : 9.9
BEGIN
NETWORK
TITLE = Init flags
      NOP   0;
//-System-------------------------------
      CLR;
      =     "SYS_infLog0";
      SET;
      =     "SYS_infLog1";
      L     0;
      T     "PLC_SystemDB".Hardware;	// Hardware ok
      L     W#16#FFFF;
      T     "PLC_SystemDB".HardwareStop;	// Hardware stop 
      L     0;
      T     "PLC_SystemDB".GlobalFlags;	// Global flags
//-Simulation with DB-------------------//[3.2]
      SET;	//[3.2]
      =     M 11.1;	//[3.2]
//-Engineering--------------------------
      SET;
      =     M 50.0;
//-Test---------------------------------
      L     0;
      T     "PLC_SystemDB".TestFunctions;	// Testfunctions
      A     "PLC_SystemDB".Startup.CmdStartTestMode;
      =     "PLC_SystemDB".GlobalFlags.StaTest;
      R     "PLC_SystemDB".Startup.CmdStartTestMode;
NETWORK
TITLE = Delay machines start after plc startup
      CLR;
      L     S5T#0MS;
      SD    T 10;
      SET;
      L     "ASW_TimerSettings".Timer10;
      SD    T 10;
NETWORK
TITLE = Init RS485 communications
      A     M 50.0;
//-> Activate or insert for every used loop the load of the value
//   Delete therefor the comment mark //
      =     M 50.0;
//      L     100
//      T     DB91.DBW   16
//      L     100
//      T     DB92.DBW   16
NETWORK
TITLE = CN Init prozess lines for coldstart/newstart
      A     "PLC_SystemDB".Startup.CmdNewstartMan;
      O     "PLC_SystemDB".Startup.CmdNewstartAuto;
      O     "PLC_SystemDB".Startup.CmdColdstartMan;
      O     "PLC_SystemDB".Startup.CmdColdstartAuto;
      JCN   CN00;
      CALL  "SYS_CallLineSection" (
           $1                       := 1);
CN00: NOP   0;
NETWORK
TITLE = WS Init prozess lines for warmstart
      A     "PLC_SystemDB".Startup.CmdRestartMan;
      O     "PLC_SystemDB".Startup.CmdRestartAuto;
      JCN   WS00;
      CALL  "SYS_CallLineSection" (
           $1                       := 2);
WS00: NOP   0;
NETWORK
TITLE = End of block
      BE;
END_FUNCTION

FUNCTION "SYS_GeneralFunctions" : VOID	// FC 105
TITLE = General plant signals
//
//COPYRIGHT:      (C) 2000 BY  BUHLER LTD.
//                           CH-9240 UZWIL  SWITZERLAND
//
//PRODUCT:        GEN_MU664
//
//TITLE:          GENERAL PLANT SIGNALS
//
//                GENERELLE ANLAGENINFORMATIONEN
//
//
//--------------------------------------------------------------------------------
//
//IDENT:          AUTOR:            DEPT:                              DATE:
//
//GEN_FC105.3.0   Ph. Engler        MU664                              05-Mar-2003
//                Redesign GCS7 Release 2
//GEN_FC105.2.0   Ph. Engler        MU664                              18-Oct-2002
//                On-Off Handling with 32-Bit and FC122
//GEN_FC105.1B    Ph. Engler        MU664                              26-May-2000
//                On-Off Handling without scratch flags
//GEN_FC105.1A    Ph. Engler        MU664                              05-Jan-2000
//                1st Release
//
//--------------------------------------------------------------------------------
//
//PURPOSE:      
//
//RESTRICTIONS: 
//
//--------------------------------------------------------------------------------
//
//
AUTHOR : PE
FAMILY : GEN
VERSION : 9.9
VAR_TEMP
  tmpBool : BOOL ;
  tmpWord : WORD ;
  tmpDWord : DWORD ;
END_VAR
BEGIN
NETWORK
TITLE = !!! Engineering remark, delete this segment !!!
      A     M 50.0;
//-> Check all input addresses in this block
//-> and delete the whole segment 1
      =     M 50.0;
      SET;
      R     "PLC_SystemDB".HardwareStop.General;
      BEU;
NETWORK
TITLE = Control voltage
      A     I 4.0;	// G_C_VOLTAGE.inp
      =     "PLC_SystemDB".Hardware.VoltageOk;
NETWORK
TITLE = Emergency stop
      A     I 4.3;	// G_ES_GENERAL.inp
      =     "PLC_SystemDB".Hardware.EsGeneralOk;
NETWORK
TITLE = Power supply motor contactor panels
      A     I 63.6;	// G_POWER_M10.inp
      =     "PLC_SystemDB".Hardware.PowerOk;
NETWORK
TITLE = Mini circuit breakers
      A     I 4.1;	// G_FUSE.inp
      =     "PLC_SystemDB".Hardware.FuseOk;
//-Delay LOG entrys in queue after fuse tripped---
      A     M 50.0;
//-> Add the following statement
      =     M 50.0;
//      UN    "GxxxG".G_FUSE.InLocal
      AN    "PLC_SystemDB".Hardware.FuseOk;
      L     "ASW_TimerSettings".Timer13;
      SE    T 13;
// 
      A     T 13;
      =     M 11.2;
NETWORK
TITLE = PLC failure
      SET;
      =     "PLC_SystemDB".Hardware.PlcOk;
NETWORK
TITLE = Fire alarms
      SET;
      =     "PLC_SystemDB".Hardware.FireOk;
NETWORK
TITLE = Smoke alarms
      SET;
      =     "PLC_SystemDB".Hardware.SmokeOk;
NETWORK
TITLE = Explosions flaps
      SET;
      =     "PLC_SystemDB".Hardware.ExflapsOk;
NETWORK
TITLE = HW-Stop
      A     "PLC_SystemDB".Hardware.VoltageOk;
      A     "PLC_SystemDB".Hardware.EsGeneralOk;
      A     "PLC_SystemDB".Hardware.PowerOk;
      A     "PLC_SystemDB".Hardware.PlcOk;
      A     "PLC_SystemDB".Hardware.FireOk;
      A     "PLC_SystemDB".Hardware.SmokeOk;
      A     "PLC_SystemDB".Hardware.ExflapsOk;
      A     T 10;
      L     "ASW_TimerSettings".Timer11;
      SD    T 11;
      AN    T 11;
      =     "PLC_SystemDB".HardwareStop.General;
NETWORK
TITLE = Section StaOffline 
      A     M 50.0;
//-> Check the input addresses
      =     M 50.0;
      NOP   0;
//-Handled from the panel front buttons---
      A     I 301.4;	// Input execute
      A     I 301.3;	// Input reset line
      L     "ASW_TimerSettings".Timer14;
      SD    T 14;
// 
//-After newstart---
      A     T 10;
      L     "ASW_TimerSettings".Timer15;
      SE    T 15;
NETWORK
TITLE = End of block
      BE;
END_FUNCTION

FUNCTION "TEST_Functions" : WORD	// FC 111
TITLE = Test functions
//
//COPYRIGHT:     (C) 2000 BY  BUHLER LTD.
//                            CH-9240 UZWIL  SWITZERLAND
//
//PRODUCT:       MELE_SMU01_99
//
//TITLE:         Test functions and simulation
//
//               Testfunktionen und Simulationen
//
// 
//--------------------------------------------------------------------------------
//
//IDENT:         AUTOR:              DEPT:                             DATE:
//
//P01_FC111.1.0  E. Hanselmann       MU664                             05-Jan-2000
//               1st Release
//
//--------------------------------------------------------------------------------
//
//PURPOSE:      
//
//RESTRICTIONS:
//
//--------------------------------------------------------------------------------
//
//
AUTHOR : EH
FAMILY : USW
VERSION : 9.9
VAR_INPUT
  code_no : INT ;	//code number
END_VAR
VAR_OUTPUT
  RET_VAL : WORD ;	//return value
END_VAR
BEGIN
NETWORK
TITLE = T00 Temporary functions (0000)
      L     #code_no;
      L     0;
      <>I;
      JC    T000;
      BEU;
T000: NOP   0;
NETWORK
TITLE = T11........................... (1001)
      L     #code_no;
      L     1001;
      <>I;
      JC    T110;
      BEU;
T110: NOP   0;
NETWORK
TITLE = T12.......................... (1002)
      L     #code_no;
      L     1002;
      <>I;
      JC    T120;
      BEU;
T120: NOP   0;
NETWORK
TITLE = T21.......................... (2001)
      L     #code_no;
      L     2001;
      <>I;
      JC    T210;
      BEU;
T210: NOP   0;
NETWORK
TITLE = T22.......................... (2002)
      L     #code_no;
      L     2002;
      <>I;
      JC    T220;
      BEU;
T220: NOP   0;
NETWORK
TITLE = End of block
      BE;
END_FUNCTION

FUNCTION "STD_LineSecStdSub" : VOID	// FC 120
TITLE = Line and section control standard subroutines
//COPYRIGHT:    (C) 2003 BY  BUHLER LTD.
//                           CH-9240 UZWIL  SWITZERLAND
//
//PRODUCT:      STD_GP    
//
//TITLE:        Line and section control standard subroutines
//              
//              Standardfunktionen für Linien und Sektionen              
//              
//
//--------------------------------------------------------------------------------
//
//IDENT:        AUTOR:              DEPT:                              DATE:
//STD_FC120.2.1 Ph.Engler           MU664                              26-May-2003
//              - Addresses of the Line parameter flags corrected
//STD_FC120.2.0 A.Egli              CT3                                18-Oct-2002
//              - New release
//STD_FC120.1.12Ph. Engler          MU664                              23-Aug-2002
//              - Function (4,1) added: Search group manual mode
//STD_FC120.1.11Ph. Engler          MU664                              30-Apr-2002
//              - Function (1,55) and (2,55) modified: Stopping/Stopped
//STD_FC120.1.10Ph. Engler          MU664                              21-Mar-2002
//              - Function (2,55): starting until S.ToSSW.infStarted
//STD_FC120.1.9 Ph. Engler          MU664                              12-Mar-2002
//              Status codes for WinCoS implemented:
//              - General group colour code
//              - Line and Section info code
//STD_FC120.1.8 Ph. Engler          MU664                              20-Mar-2001
//              Line status colour for 2-4 section implemented
//STD_FC120.1.7 Ph. Engler          MU664                              20-Dec-2000
//              Pre stop weight for cmdSequenceStop
//STD_FC120.1.6 Ph. Engler          MU664                              14-Dec-2000
//              - Substitude Bincode into recipe extended, InCode 3 
//              - JS Job paramter flags (2,2) Sta-Address corrected
//STD_FC120.1.5 Ph. Engler          MU664                              01-Nov-2000
//              CmdSequenceStop only if section is in StActive           
//STD_FC120.1.4 Ph. Engler          MU664                              19-Okt-2000
//              Update SND-Binlist staSameSndRcv:
//               Suppression of the error meassage 'bin not found'
//STD_FC120.1.3 Ph. Engler          MU664                              28-Jun-2000
//              Section text and colour code extension 
//              with code 702, 703 and 1402
//STD_FC120.1.2 Ph. Engler          MU664                              04-May-2000
//              LS Line state/fault protocolling (1,10)
//               esXXX corrected 
//STD_FC120.1.1 Ph. Engler          MU664                              29-Mar-2000
//              Line log messages implemented
//STD_FC120.1.0 Ph. Engler          MU664                              05-Jan-2000
//              1st Release
//
//--------------------------------------------------------------------------------
//
//PURPOSE:      These function are callt by Line Control and
//              Section Control.
//              The most subroutine are handled by FB90
//
//RESTRICTIONS:
//
//--------------------------------------------------------------------------------
//
//InCode: 
//1000 to 1999: Subroutines Line
//              For Input and Output parameter is 
//              LineDB.VarTemp used  
//2000 to 2999: Subroutines Section
//              For Input and Output parameter is
//              SectionDB.VarTemp used  
//
//
//
//
AUTHOR : PE
FAMILY : STD
VERSION : 2.0
VAR_INPUT
  InCode : INT ;	//Code number; 1000=Line 2=Section
END_VAR
BEGIN
NETWORK
TITLE = Sub1031: CF Clear line flags 
//Open DB=  Line Parameter DB
      L     #InCode;
      L     1031;
      <>I;
      JC    CF00;
//Line parameter DB
      L     L#0;
      T     DBD 300;	// Section 1
      T     DBD 304;	// Section 2
      T     DBD 308;	// Section 3
      T     DBD 312;	// Section 4
      T     DBD 316;	// General
      T     DBD 320;	// General
CF00: NOP   0;
NETWORK
TITLE = All other Subroutines are handled by FB90
      CDB;
      L     #InCode;
      T     DIW 0;	//InCode
//-Call Methode FB90---
      UC    "STD_LineSecStdSub2";
NETWORK
TITLE = End of block
      BE;
END_FUNCTION

FUNCTION "STD_OnOffSignals32" : VOID	// FC 122
TITLE = FKT: ON / OFF Signal handling
//COPYRIGHT:      (C) 2000 BY  BUHLER LTD.
//                           CH-9240 UZWIL  SWITZERLAND
//
//PRODUCT:        STD_MU664
//
//TITLE:          ON / OFF Signal handling
//                  32-Bit
//                ON / OFF Signal Hantierung
//                  32-Bit
//
//--------------------------------------------------------------------------------
//
//IDENT:          AUTOR:            DEPT:                              DATE:
//
//STD_FC122.1.0   Ph. Engler        MU664                              18-Oct-2002
//                1st Release
//
//--------------------------------------------------------------------------------
//
//PURPOSE:      
//
//RESTRICTIONS: 
//
//--------------------------------------------------------------------------------
//
//
AUTHOR : PE
FAMILY : STD
VERSION : 0.0
VAR_INPUT
  InCodeNo : INT ;	//Selection of function
  MaskUsedBits : DWORD ;	//Number of used bits
END_VAR
VAR_IN_OUT
  cmdOn : DWORD ;	//Command to set the status
  cmdOff : DWORD ;	//Command to reset the status
  staOn : DWORD ;	//Status
  cmdChanged : BOOL ;	//Pulse if status changed
END_VAR
VAR_TEMP
  staSaved : DWORD ;	//Saved status
END_VAR
BEGIN
NETWORK
TITLE = SS Save status
//The status of not selected bits will be saved.
      L     #staOn;
      L     #MaskUsedBits;
      INVD;
      AD;
      T     #staSaved;
NETWORK
TITLE = PS Pulse signal
      L     #InCodeNo;
      L     1;
      <>I;
      JC    PS00;
      L     #cmdOn;	// ( Only selected bits
      L     #MaskUsedBits;	// ( 
      AD;	// (
      L     #staSaved;	//  ( Restore not selected bits
      OD;	//  (
      T     #staOn;	// ( Save pulse
      L     #MaskUsedBits;	//  ( Reset on commands 
      INVD;	//  (
      L     #cmdOn;	//  (
      AD;	//  (
      T     #cmdOn;	//  (
      L     #MaskUsedBits;	// ( Reset off commands 
      INVD;	// (
      L     #cmdOff;	// (
      AD;	// (
      T     #cmdOff;	// (
      BEU;
PS00: NOP   0;
NETWORK
TITLE = SS Status signal
//Use this cmdChanged pulse to go trough the group preselection again.
      L     #InCodeNo;
      L     2;
      <>I;
      JC    SS00;
//-Detect new commands------------------
      A(;	// (
      L     #staOn;	// ( Check change to on
      INVD;	// (
      L     #cmdOn;	// (
      AD;	// (
      L     #MaskUsedBits;	// ( 
      AD;	// (
      L     0;	// (
      <>D;	// (
      );	// (
      O(;	//  (
      L     #staOn;	//  ( Check change to off
      L     #cmdOff;	//  (
      AD;	//  (
      L     #MaskUsedBits;	//  ( 
      AD;	//  (
      L     0;	//  (
      <>D;	//  (
      );	//  (
      =     #cmdChanged;	// ( --> Set signal
//-Update status------------------------
      L     #staOn;	// ( Set status
      L     #cmdOn;	// (
      OD;	// (
      L     #cmdOff;	//  ( Reset status
      INVD;	//  (
      AD;	//  (
      L     #MaskUsedBits;	// ( Save only selected bits
      AD;	// (
      L     #staSaved;	//  ( Restore not selected bits
      OD;	//  (
      T     #staOn;	// ( Save status
      L     #MaskUsedBits;	//  ( Reset on commands 
      INVD;	//  (
      L     #cmdOn;	//  (
      AD;	//  (
      T     #cmdOn;	//  (
      L     #MaskUsedBits;	// ( Reset off commands 
      INVD;	// (
      L     #cmdOff;	// (
      AD;	// (
      T     #cmdOff;	// (
      BEU;
SS00: NOP   0;
NETWORK
TITLE = End of block
      BE;
END_FUNCTION

FUNCTION "COM_PLCtoPLC" : VOID	// FC 141
TITLE = PLC to PLC Communication
//COPYRIGHT:    (C) 2003  BUHLER AG, CH-9240 UZWIL, SWITZERLAND
//
//PRODUCT:      ZZZZ_ZZZ01_00
//
//TITLE:        PLC to PLC Communication
//                 Prepare communication data
//              SPS zu SPS Kommunikation
//                 Datenaufbereitung
//
//--------------------------------------------------------------------------------
//
//IDENT:        AUTHOR:             DEPT:                              DATE:
//
//P0x_FC141.2.0 Ph. Engler          MU664                              02-Feb-2003
//              Redesign GCS7 Release 2
//P0x_FC141.1.0 Ph. Engler          MU664                              13-Dec-2000
//              1st release
//
//--------------------------------------------------------------------------------
//
//PURPOSE:      
//
//MANUAL : GRMENMEN.DOC
//
//RESTRICTIONS: S7
//
//--------------------------------------------------------------------------------
//
AUTHOR : PE
FAMILY : USW
VERSION : 9.9
VAR_TEMP
  Var1 : DINT ;
END_VAR
BEGIN
NETWORK
TITLE = P1 Communication with PLC1
      A     M 50.0;	// Check if communication is needed
      JC    P100;
      A     DB131.DBX 59.3;
      JC    P100;
// 
//-Send data to PLC1---
      A     M 50.0;
//-> Create the data buffer DB1761 as an instanz db for FB701
//-> Correct Len_SendData depends on data to send, for MPI communication the minimum as possible
      =     M 50.0;
      CALL  FB 1701 , "ComPLC1Snd" (
           DIW 0                    := 1809,
           DIW 2                    := 1711,
           DIW 4                    := 0,
           DIW 6                    := 200,
           DIW 8                    := 10,
           DIW 10                   := 5);	// [Bytes]
// 
//-Clear commands---
      A     M 50.0;
//-> Reset the following commands for each transmitted virtual/imported group
//   Y = PLCNo of the real group
//   x = Number of the group
      =     M 50.0;
//      U     "ComPLC1Snd".CmdCopied
//      R     "ComPLC1Snd".CmdCopied
//      R     "PLC1Snd".GrYxxx.CmdFaultReset
//      R     "PLC1Snd".GrYxxx.CmdNext
//      R     "PLC1Snd".GrYxxx.CmdManualOff
//      R     "PLC1Snd".GrYxxx.CmdNewJob
//      R     "PLC1Snd".GrYxxx.CmdNewValue
//      R     "PLC1Snd".GrYxxx.CmdRestartIdling
// 
//-Receive data form PLC1---
      A     M 50.0;
//-> Create the data buffer DB1771 as an instanz db for FB702
//-> Correct Len_SendData depends on data to send, for MPI communication the minimum as possible
      =     M 50.0;
      CALL  FB 1702 , "ComPLC1Rcv" (
           DIW 0                    := 1825,
           DIW 2                    := 1721,
           DIW 4                    := 0,
           DIW 6                    := 200,
           DIW 8                    := 20);	// [Bytes]
P100: NOP   0;
NETWORK
TITLE = P2 Communication with PLC2
      A     M 50.0;	// Check if communication is needed
      JC    P200;
      A     DB132.DBX 59.3;
      JC    P200;
// 
//-Send data to PLC2---
      A     M 50.0;
//-> Create the data buffer DB1762 as an instanz db for FB701
//-> Correct Len_SendData depends on data to send, for MPI communication the minimum as possible
      =     M 50.0;
      CALL  FB 1701 , "ComPLC2Snd" (
           DIW 0                    := 1810,
           DIW 2                    := 1712,
           DIW 4                    := 0,
           DIW 6                    := 200,
           DIW 8                    := 10,
           DIW 10                   := 5);	// [Bytes]
// 
//-Clear commands---
      A     M 50.0;
//-> Reset the following commands for each transmitted virtual/imported group
//   Y = PLCNo of the real group
//   x = Number of the group
      =     M 50.0;
//      U     "ComPLC2Snd".CmdCopied
//      R     "ComPLC2Snd".CmdCopied
//      R     "PLC2Snd".GrYxxx.CmdFaultReset
//      R     "PLC2Snd".GrYxxx.CmdNext
//      R     "PLC2Snd".GrYxxx.CmdManualOff
//      R     "PLC2Snd".GrYxxx.CmdNewJob
//      R     "PLC2Snd".GrYxxx.CmdNewValue
//      R     "PLC2Snd".GrYxxx.CmdRestartIdling
// 
//-Receive data form PLC2---
      A     M 50.0;
//-> Create the data buffer DB1772 as an instanz db for FB702
//-> Correct Len_SendData depends on data to send, for MPI communication the minimum as possible
      =     M 50.0;
      CALL  FB 1702 , "ComPLC2Rcv" (
           DIW 0                    := 1826,
           DIW 2                    := 1722,
           DIW 4                    := 0,
           DIW 6                    := 200,
           DIW 8                    := 20);	// [Bytes]
P200: NOP   0;
NETWORK
TITLE = P3 Communication with PLC3
      A     M 50.0;	// Check if communication is needed
      JC    P300;
      A     DB133.DBX 59.3;
      JC    P300;
// 
//-Send data to PLC3---
      A     M 50.0;
//-> Create the data buffer DB1763 as an instanz db for FB701
//-> Correct Len_SendData depends on data to send, for MPI communication the minimum as possible
      =     M 50.0;
      CALL  FB 1701 , "ComPLC3Snd" (
           DIW 0                    := 1811,
           DIW 2                    := 1713,
           DIW 4                    := 0,
           DIW 6                    := 200,
           DIW 8                    := 10,
           DIW 10                   := 5);	// [Bytes]
// 
//-Clear commands---
      A     M 50.0;
//-> Reset the following commands for each transmitted virtual/imported group
//   Y = PLCNo of the real group
//   x = Number of the group
      =     M 50.0;
//      U     "ComPLC3Snd".CmdCopied
//      R     "ComPLC3Snd".CmdCopied
//      R     "PLC3Snd".GrYxxx.CmdFaultReset
//      R     "PLC3Snd".GrYxxx.CmdNext
//      R     "PLC3Snd".GrYxxx.CmdManualOff
//      R     "PLC3Snd".GrYxxx.CmdNewJob
//      R     "PLC3Snd".GrYxxx.CmdNewValue
//      R     "PLC3Snd".GrYxxx.CmdRestartIdling
// 
//-Receive data form PLC3---
      A     M 50.0;
//-> Create the data buffer DB1773 as an instanz db for FB702
//-> Correct Len_SendData depends on data to send, for MPI communication the minimum as possible
      =     M 50.0;
      CALL  FB 1702 , "ComPLC3Rcv" (
           DIW 0                    := 1827,
           DIW 2                    := 1723,
           DIW 4                    := 0,
           DIW 6                    := 200,
           DIW 8                    := 20);	// [Bytes]
P300: NOP   0;
NETWORK
TITLE = P4 Communication with PLC4
      A     M 50.0;	// Check if communication is needed
      JC    P400;
      A     DB134.DBX 59.3;
      JC    P400;
// 
//-Send data to PLC4---
      A     M 50.0;
//-> Create the data buffer DB1764 as an instanz db for FB701
//-> Correct Len_SendData depends on data to send, for MPI communication the minimum as possible
      =     M 50.0;
      CALL  FB 1701 , "ComPLC4Snd" (
           DIW 0                    := 1812,
           DIW 2                    := 1714,
           DIW 4                    := 0,
           DIW 6                    := 200,
           DIW 8                    := 10,
           DIW 10                   := 5);	// [Bytes]
// 
//-Clear commands---
      A     M 50.0;
//-> Reset the following commands for each transmitted virtual/imported group
//   Y = PLCNo of the real group
//   x = Number of the group
      =     M 50.0;
//      U     "ComPLC4Snd".CmdCopied
//      R     "ComPLC4Snd".CmdCopied
//      R     "PLC4Snd".GrYxxx.CmdFaultReset
//      R     "PLC4Snd".GrYxxx.CmdNext
//      R     "PLC4Snd".GrYxxx.CmdManualOff
//      R     "PLC4Snd".GrYxxx.CmdNewJob
//      R     "PLC4Snd".GrYxxx.CmdNewValue
//      R     "PLC4Snd".GrYxxx.CmdRestartIdling
// 
//-Receive data form PLC4---
      A     M 50.0;
//-> Create the data buffer DB1774 as an instanz db for FB702
//-> Correct Len_SendData depends on data to send, for MPI communication the minimum as possible
      =     M 50.0;
      CALL  FB 1702 , "ComPLC4Rcv" (
           DIW 0                    := 1828,
           DIW 2                    := 1724,
           DIW 4                    := 0,
           DIW 6                    := 200,
           DIW 8                    := 20);	// [Bytes]
P400: NOP   0;
NETWORK
TITLE = P5 Communication with PLC5
      A     M 50.0;	// Check if communication is needed
      JC    P500;
      A     DB135.DBX 59.3;
      JC    P500;
// 
//-Send data to PLC5---
      A     M 50.0;
//-> Create the data buffer DB1765 as an instanz db for FB701
//-> Correct Len_SendData depends on data to send, for MPI communication the minimum as possible
      =     M 50.0;
      CALL  FB 1701 , "ComPLC5Snd" (
           DIW 0                    := 1813,
           DIW 2                    := 1715,
           DIW 4                    := 0,
           DIW 6                    := 200,
           DIW 8                    := 10,
           DIW 10                   := 5);	// [Bytes]
// 
//-Clear commands---
      A     M 50.0;
//-> Reset the following commands for each transmitted virtual/imported group
//   Y = PLCNo of the real group
//   x = Number of the group
      =     M 50.0;
//      U     "ComPLC5Snd".CmdCopied
//      R     "ComPLC5Snd".CmdCopied
//      R     "PLC5Snd".GrYxxx.CmdFaultReset
//      R     "PLC5Snd".GrYxxx.CmdNext
//      R     "PLC5Snd".GrYxxx.CmdManualOff
//      R     "PLC5Snd".GrYxxx.CmdNewJob
//      R     "PLC5Snd".GrYxxx.CmdNewValue
//      R     "PLC5Snd".GrYxxx.CmdRestartIdling
// 
//-Receive data form PLC5---
      A     M 50.0;
//-> Create the data buffer DB1775 as an instanz db for FB702
//-> Correct Len_SendData depends on data to send, for MPI communication the minimum as possible
      =     M 50.0;
      CALL  FB 1702 , "ComPLC5Rcv" (
           DIW 0                    := 1829,
           DIW 2                    := 1725,
           DIW 4                    := 0,
           DIW 6                    := 200,
           DIW 8                    := 20);	// [Bytes]
P500: NOP   0;
NETWORK
TITLE = End of block
      BE;
END_FUNCTION

FUNCTION "STD_SearchChangeBit" : VOID	// FC 241
TITLE = Search object change bits
//COPYRIGHT:    (C) 2000 BY  BUEHLER LTD.
//                           CH-9240 UZWIL  SWITZERLAND
//
//PRODUCT:      STD_MU664
//
//TITLE:        Search object change bits
//
//              Suchen der Change Bits eines Objektes
//
//
//--------------------------------------------------------------------------------
//
//IDENT:        AUTOR:              DEPT:                              DATE:
//
//STD_FC241.1.0 Ph. Engler          MU664                              26-May-2000
//              1st Release
//
//--------------------------------------------------------------------------------
//
//PURPOSE:      
//
//RESTRICTIONS: S7
//
//--------------------------------------------------------------------------------
//
AUTHOR : PE
FAMILY : STD
VERSION : 0.0
VAR_INPUT
  ChangeBitDBNr : BLOCK_DB ;	//Datablock of the change bit interface
  ObjectDBNr : INT ;	//Datablock number of the object
END_VAR
VAR_OUTPUT
  CBit1 : BOOL ;	//Change bit 1
  CBit2 : BOOL ;	//Change bit 2
  CBit3 : BOOL ;	//Change bit 3
  CBit4 : BOOL ;	//Change bit 4
  ObjectFound : BOOL ;	//Datablock of requested object was found in the change bit data block
END_VAR
VAR_TEMP
  TmpLoopCounterInitValue : INT ;
  TmpLoopCounter : INT ;
  TmpAddressRegInitValue : DWORD ;
  TmpAddressReg : DWORD ;
END_VAR
BEGIN
NETWORK
TITLE = LI Loop initial value calculation
      OPN   #ChangeBitDBNr;	// Call change bit data block
      L     DBLG;	// Length of change bit data block
      L     DBW 10;	// ParDWCopyBits
      ITD;	// 
      -D;	// 
      +     -160;	// Offset pointer table
      L     4;	// 
      /D;	// 
      +     -1;	// 
      T     #TmpLoopCounterInitValue;	// => Loop init
NETWORK
TITLE = AI Address register initial value calculation
      OPN   #ChangeBitDBNr;	// Call change bit data block
      L     DBW 10;	// ParDWCopyBits
      +     160;	// Offset pointer table
      SLD   3;	// Byte to bit-adress (x8)
      T     #TmpAddressRegInitValue;	// => Init address
      T     #TmpAddressReg;	// => Init bit-adress
NETWORK
TITLE = SC Search change bit
      L     #TmpLoopCounterInitValue;	// 
SC01: T     #TmpLoopCounter;	// 
      OPN   #ChangeBitDBNr;	// Call change bit data block
      L     DBW [#TmpAddressReg];	// 
      L     #ObjectDBNr;	// 
      ==I;	// Compare data block numbers
      JC    SC02;	// If equal then found
//-Next loop---
      L     #TmpAddressReg;	// Bit-adress
      +     32;	// Increment 32 bit (DWORD)
      T     #TmpAddressReg;	// => Bit-adress
      L     #TmpLoopCounter;	// 
      LOOP  SC01;	// 
//-Not found---
      CLR;
      =     #ObjectFound;
      JU    SC00;
//-Found---
SC02: L     #TmpAddressReg;
      L     #TmpAddressRegInitValue;
      -D;	//number of bit until found
      L     32;
      /D;	//number of pointer DBD
      L     4;
      *D;	//bit number c-bit area
      L     P#200.0;	//offset begin c-bit area
      +D;
      LAR1;
      OPN   #ChangeBitDBNr;	// Call change bit data block
      A     DBX [AR1,P#0.0];	// 
      =     #CBit1;	// => Change bit 1
      A     DBX [AR1,P#0.1];	// 
      =     #CBit2;	//  => Change bit 2
      A     DBX [AR1,P#0.2];	// 
      =     #CBit3;	// => Change bit 3
      A     DBX [AR1,P#0.3];	// 
      =     #CBit4;	//  => Change bit 4
      SET;
      =     #ObjectFound;
SC00: NOP   0;
NETWORK
TITLE = End of block
      BE;
END_FUNCTION

FUNCTION "STD_PLCLiveValue" : VOID	// FC 242
TITLE = Live value handling for PCC
//COPYRIGHT:    (C) 2000 BY  BUEHLER LTD.
//                           CH-9240 UZWIL  SWITZERLAND
//
//PRODUCT:      STD_MU664
//
//TITLE:        Live value handling for PCC
//
//              Aufbereitung des Lebenssignals für das Leitsystem
//
//
//--------------------------------------------------------------------------------
//
//IDENT:        AUTOR:              DEPT:                              DATE:
//
//STD_FC242.1B  Ph. Engler          MU664                              16-Sep-2004
//              Counter speed increased from 1sec to 200ms
//STD_FC242.1A  Ph. Engler          MU664                              19-Okt-2000
//              1st Release
//
//--------------------------------------------------------------------------------
//
//PURPOSE:      
//
//RESTRICTIONS: S7
//
//--------------------------------------------------------------------------------
//
AUTHOR : PE
FAMILY : STD
VERSION : 0.0
VAR_IN_OUT
  LiveValue : INT ;	//Dataword of the lifevalue from a changebit datablock
END_VAR
BEGIN
NETWORK
TITLE = IC Increment counter
      A     "SYS_Scan0_Tick200ms";
      JCN   IC00;
      L     #LiveValue;
      L     1;
      +I;
      T     #LiveValue;
IC00: NOP   0;
NETWORK
TITLE = End of block
      BE;
END_FUNCTION

FUNCTION "STD_AuxiliaryFunctions" : VOID	// FC 247
TITLE = Auxiliary functions
//COPYRIGHT:    (C) 2000 BY  BUEHLER LTD.
//                           CH-9240 UZWIL  SWITZERLAND
//
//PRODUCT:      STD_MU664
//
//TITLE:        Auxiliary functions
//
//              Hilfsfunktionen
//
//
//--------------------------------------------------------------------------------
//
//IDENT:        AUTOR:              DEPT:                              DATE:
//
//STD_FC247.1.0 Ph. Engler          MU664                              05-Jan-2000
//              1st Release
//
//--------------------------------------------------------------------------------
//
//PURPOSE:      -
//
//RESTRICTIONS: - S7
//
//--------------------------------------------------------------------------------
//
AUTHOR : PE
FAMILY : STD
VERSION : 0.0
VAR_INPUT
  InFctNo : INT ;	//Function number
  InPointer : DWORD ;
  InInt1 : INT ;
  InInt2 : INT ;
END_VAR
VAR_OUTPUT
  OutInt1 : INT ;
  OutInt2 : INT ;
END_VAR
VAR_TEMP
  TmpLoop1Counter : INT ;
  TmpLoop2Counter : INT ;
END_VAR
BEGIN
NETWORK
TITLE = CB Count number of bit in any range
//inPointer = Bit-Startaddress as pointer, ie P#M 100.0
//inInt1    = Number of byte from start address
//outInt1   = Number of high bit
      L     #InFctNo;
      L     1;
      ==I;
      JCN   CB00;
      NOP   0;
//-Init---
      L     #InPointer;
      LAR1;
      L     0;
      T     #OutInt1;
//-Count number of bits set---
      L     #InInt1;
LOP1: T     #TmpLoop1Counter;
      L     8;	// Number of bits
LOP2: T     #TmpLoop2Counter;
      A      [AR1,P#0.0];	// Read actual bit
      JCN   NEXT;
      L     #OutInt1;
      INC   1;
      T     #OutInt1;
NEXT: +AR1  P#0.1;
      L     #TmpLoop2Counter;
      LOOP  LOP2;	// Bit counter
      L     #TmpLoop1Counter;
      LOOP  LOP1;	// Byte counter
CB00: NOP   0;
NETWORK
TITLE = MM Search min/max values
//inPointer = Word-Startaddress as pointer, ie P#M 2000.0
//inInt1    = Number of words from start address, with values to check
//outInt1   = MinValue
//outInt2   = MaxValue
      L     #InFctNo;
      L     2;
      ==I;
      JCN   MM00;
//-Init variables---
      L     0;	// )
      T     #OutInt2;	// ) Max value
      L     W#16#7FFF;	//  )
      T     #OutInt1;	//  ) Min value
      L     #InPointer;	//  )
      LAR1;	//  ) Address register 1
      L     #InInt1;	// ) 
//-Max value---
MM01: T     #TmpLoop1Counter;	// ) Loop counter
      L     W [AR1,P#0.0];	// ) Load new value
      L     #OutInt2;	// ) Max value
      >=I;	// ) If new value >= max value then
      JCN   MM02;	// ) 
      TAK;	// )
      T     #OutInt2;	// ) --> Save new value
//-Min value---
MM02: L     W [AR1,P#0.0];	// ) Load new value
      L     #OutInt1;	// ) Min value
      <=I;	// ) If new value <= min value then
      JCN   MM03;	// ) 
      TAK;	// )
      T     #OutInt1;	// ) --> Save new value
//-Loop---
MM03: +AR1  P#2.0;
      L     #TmpLoop1Counter;
      LOOP  MM01;
MM00: NOP   0;
NETWORK
TITLE = End of block
      BE;
END_FUNCTION

FUNCTION "STD_EdgeFunctions" : VOID	// FC 248
TITLE = STD: Edge / step functions
//COPYRIGHT:    (C) 2004 BY  BUEHLER LTD.
//                           CH-9240 UZWIL  SWITZERLAND
//
//PRODUCT:      STD_MU664
//
//TITLE:        EDGE/STEP FUNCTIONS
//
//              FLANKEN/SCHRITT FUNKTIONEN
//
//
//--------------------------------------------------------------------------------
//
//IDENT:        AUTOR:              DEPT:                              DATE:
//
//STD_FC248.1.0 Ph. Engler          MU664                              7-May-2004
//              1st Release
//
//--------------------------------------------------------------------------------
//
//PURPOSE:      -
//
//RESTRICTIONS: - S7
//
//--------------------------------------------------------------------------------
//
//PURPOSE:      - Bildet aus dem Eingangssignal ein Schrittsignal,
//                eine positive und eine negative Flanke (Wortweise).
//
//RESTRICTIONS: - Die Uebergabeparameter koennen EW, AW, MW oder DW
//                (vom aufgeschlagenen DB) sein.
//
//--------------------------------------------------------------------------------
//
AUTHOR : PE
FAMILY : STD
VERSION : 1.0
VAR_INPUT
  INP : WORD ;	// INP
END_VAR
VAR_OUTPUT
  HS : WORD ;	// HS
  POS : WORD ;	// POS
  NEG : WORD ;	// NEG
  STEP : WORD ;	// STEP
END_VAR
BEGIN
NETWORK
TITLE =
//Funktionen:
//===========
//
//STEP  - Wechselt bei jeder positiven Flanke des Eingangsignals (INP)
//        seinen Zustand (Log. 0 -> 1  /  1 -> 0).
//POS   - Wechselt bei jeder positiven Flanke des Eingangsignals (INP)
//        waehrend einem Programmzyklus seinen Zustand von Log. 0 nach 1.
//NEG   - Wechselt bei jeder negativen Flanke des Eingangsignals (INP)
//        waehrend einem Programmzyklus seinen Zustand von Log. 0 nach 1.
//HS    - Das Hilfssignal wird zur Erkennung der positiven Flanke vom
//        Eingangssignal (INP) benoetigt (keine Schmiermerker verwenden !!).
//
//Hinweise:
//---------
//
//- Fuer STEP, POS, NEG koennen Schmiermerker verwendet werden falls
//  sie im Programm-Code nicht ausgewertet werden.
//
//- Die Abfrage   U  "POS-Bit"
//                U  "STEP-Bit"
//ergibt waehrend einem Programmzyklus eine Flanke "Schritt Ein"
//
//- Die Abfrage   U  "POS-Bit"
//                UN "STEP-Bit"
//ergibt waehrend einem Programmzyklus eine Flanke "Schritt Aus"
//
//
//       |     |   |   |      |   |   |      |   |   |      |   |   |
//     1 |     | 1--------------1 |   |      | 1--------------1 |   |
//HS   0 |-------0 |   |      | 0--------------0 |   |      | 0---------
//       |     |   |   |      |   |   |      |   |   |      |   |   |
//     1 |     |   |   |      | 1---1 |      |   |   |      | 1---1 |
//NEG  0 |----------------------0 | 0-------------------------0 | 0-----
//       |     |   |   |      |   |   |      |   |   |      |   |   |
//     1 |     | 1---1 |      |   |   |      | 1---1 |      |   |   |
//POS  0 |-------0 | 0-------------------------0 | 0--------------------
//       |     |   |   |      |   |   |      |   |   |      |   |   |
//     1 |     | 1-----------------------------1 |   |      |   |   |
//STEP 0 |-------0 |   |      |   |   |      | 0------------------------
//       |     |   |   |      |   |   |      |   |   |      |   |   |
//     1 | 1---------------1  |   |   |   1--------------1  |   |   |
//INP  0 |-0   |   |   |   0--------------0  |   |   |   0--------------
//-------|-----|---|---|------|---|---|------|---|---|------|---|---|--------
//       |     |   |   |      |   |   |      |   |   |      |   |   |
//Zykl.        1   2          1   2          1   2          1   2
//
      L     #INP;	// Eingangssignal
      L     #HS;	// Hilfssignal
      INVI;
      AW;
      T     #POS;	// Positive Flanke
      L     #STEP;	// Schrittsignal
      XOW;
      T     #STEP;	// Schrittsignal
      L     #INP;	// Eingangssignal
      INVI;
      L     #HS;	// Hilfssignal
      AW;
      T     #NEG;	// Negative Flanke
      L     #INP;
      T     #HS;	// Hilfssignal
NETWORK
TITLE = End of block
      BE;
END_FUNCTION

FUNCTION "STD_ScaleAnalogSignal" : VOID	// FC 249
TITLE = Scale S7 Analogues for S5
//COPYRIGHT:    (C) 1998 BY  BUHLER AG
//                           CH-9240 UZWIL  SWITZERLAND
//
//PRODUCT:      AME01_98
//
//TITLE:        Scale S7 Analogues for S5
//              
//
//-------------------------------------------------------------------------
//
//IDENT:        AUTHOR:             DEPT:             DATE:
//
//FC105.1A      GS                  CDDP              15-Jan-2000
//              1st Release
//
//-------------------------------------------------------------------------
//
//PURPOSE: 
//
//RESTRICTIONS: 
//
//-------------------------------------------------------------------------
//
//Functions
//=========
//
//  01 - S5 Analogue Input 0..20mA
//  02 - S5 Analogue Input 4..20mA
//  03 - S5 Analogue Output 0..20mA or 4..20mA card
//  04 - S5 Analogue Output 4..20mA on a 0..20mA card
//
//
AUTHOR : GS
FAMILY : ASW
NAME : ANA_S5_S
VERSION : 1.0
VAR_INPUT
  function_no : INT ;	//function selection
END_VAR
VAR_TEMP
  Inputvalue : INT ;
  OutputValue : INT ;
END_VAR
BEGIN
NETWORK
TITLE = Initialisation
      TAK;
      T     #Inputvalue;
NETWORK
TITLE = S5 Analogue Input 0..20mA
// (network holds code this reader does not know; not shown)
// S5 Analogue inputs cards 0..20mA give a number of 0..2048
// Bottom 3 bits are used for over/under range indication from the card
// All S7 modules use 0..27648 as 0..100%
// Conversion formula is:-
//  
//     S5Value  * 27648
//     -------
//      2048
// 
NETWORK
TITLE = S5 Analogue Input 4..20mA
// (network holds code this reader does not know; not shown)
// S5 Analogue inputs cards 4..20mA give a number of 0..2560
// but have an offset of 512. This gives 512..2560 = 4..20mA
// 2048 units cover 16mA.
// Bottom 3 bits are used for over/under range indication from the card
// All S7 modules use 0..27648 as 0..100%
// Conversion formula is:-
//  
//     (S5Value - 512)  * 27648
//     ---------------
//          2048
// 
NETWORK
TITLE = S5 Analogue Output 0..20mA or 4..20mA card
      L     #function_no;
      L     3;
      <>I;
      JC    en03;
// S5 Analogue Outputs cards use a number of 0..1024
// Bottom 4 bits are not used used
// All S7 modules use 0..27648 as 0..100%
// Conversion formula is:-
//  
//     S7Value  * 1024
//     -------
//      27648
// 
      L     #Inputvalue;
      DTR;
      L     2.764800e+04;	// 27648
      /R;
      L     1.024000e+03;	// 1024
      *R;
      RND;
      SLW   4;
      T     #OutputValue;
en03: NOP   0;
NETWORK
TITLE = S5 Analogue Output 4..20mA on a 0..20mA card
      L     #function_no;
      L     4;
      <>I;
      JC    en04;
// S5 Analogue Outputs cards use a number of 0..1024
// Bottom 4 bits are not used used
// All S7 modules use 0..27648 as 0..100%
// Conversion formula is:-
//  
//    ( S7Value  * 820 ) + 204
//      -------
//       27648
// 
// Note:   820 is 4/5ths of 1024    (for the 4..20mA portion)
//         204 is 1/5th of 1024     (for the 0..4mA portion)
// 
      L     #Inputvalue;
      DTR;
      L     2.764800e+04;	// 27648
      /R;
      L     8.200000e+02;	// 820
      *R;
      L     2.040000e+02;	// 204
      +R;
      RND;
      SLW   4;
      T     #OutputValue;
en04: NOP   0;
NETWORK
TITLE = S5 Analogue Input -20..20mA convert to 4..20mA 
//  L     #function_no
//      L     5
//      <>I   
//      SPB   en05
//
//// S5 Analogue inputs cards 0..20mA give a number of 0..2048
//// Bottom 3 bits are used for over/under range indication from the card
//// All S7 modules use 0..27648 as 0..100%
//// Conversion formula is:-
////  
////     S5Value  * 27648
////     ----------------  +  409
////           2048
//// 
//// Note:   1636 is 4/5th of approx. 2048  (for the 4..20mA portion)
////         409 is 1/5th of approx. 2048  (for the 0..4mA portion)
//// 
//
//      L     #Inputvalue
//      SSI   3                           // Shift to right with sign !
//      L     409
//      <I    
//      SPB   zer5
//      TAK   
//      DTR   
//      L     2.048000e+003               // 2048
//      /R    
//      L     2.764800e+004               // 27648
//      *R    
//      RND   
//      L     L#5535
//      -D    
//      DTR   
//      L     1.200000e+000
//      *R    
//      RND   
//      SPA   Val5
//zer5: L     0
//Val5: T     #OutputValue
//
//en05: NOP   0
//
// (network holds code this reader does not know; not shown)
// S5 Analogue inputs cards 0..20mA give a number of 0..2048
// Bottom 3 bits are used for over/under range indication from the card
// All S7 modules use 0..27648 as 0..100%
// Conversion formula is:-
//  
//     S5Value - 409
//     ----------------  *  27648 + 1.25
//           2048
// 
// Note:   1636 is 4/5th of approx. 2048  (for the 4..20mA portion)
//         409 is 1/5th of approx. 2048  (for the 0..4mA portion)
// 
NETWORK
TITLE = Output final value
      L     #OutputValue;
END_FUNCTION

DATA_BLOCK "PLC_SystemDB"	// DB 50
//COPYRIGHT:    (C) 2000 BY  BUHLER AG
//                           CH-9240 UZWIL  SWITZERLAND
//
//PRODUCT:      STD_MU664
//
//TITLE:        PLC: System informations
//
//              PLC: Systeminformationen
//
//
//--------------------------------------------------------------------------------
//
//IDENT:        AUTHOR:             DEPT:                              DATE:
//
//STD_DB050.1.1 Ph. Engler          MU664                              21-Dec-2000
//              ColdStart signals and counter integrated
//STD_DB050.1A  Ph. Engler          MU664                              05-Jan-2000
//              1st Release
//
//--------------------------------------------------------------------------------
//
//PURPOSE:  
//MANUAL : 
//CODE   :
//RESTRICTIONS:
//
//--------------------------------------------------------------------------------
//
//
//
//
//
//
//
AUTHOR : PE
FAMILY : GEN
VERSION : 9.9
  STRUCT
   Spare00 : WORD ;
   Startup : STRUCT
    CmdNewstartMan : BOOL ;	//Manual newstart active
    CmdNewstartAuto : BOOL ;	//Automatic newstart active
    CmdRestartMan : BOOL ;	//Manual restart requested
    CmdRestartAuto : BOOL ;	//Automatic restart requested
    CmdColdstartMan : BOOL ;	//Manual coldstart requested
    CmdColdstartAuto : BOOL ;	//Automatic coldstart requested
    NotUsed06 : BOOL ;
    NotUsed07 : BOOL ;
    CmdStartTestMode : BOOL ;	//Starts the test mode
   END_STRUCT ;
   StartupCounter : STRUCT
    NewstartMan : INT ;	//Number of manual newstart startups
    NewstartAuto : INT ;	//Number of automatic newstart startups
    RestartMan : INT ;	//Number of manual restart startups
    RestartAuto : INT ;	//Number of automatic restart startups
    ColdstartMan : INT ;	//Number of manual coldstart startups
    ColdstartAuto : INT ;	//Number of automatic coldstart startups
    NotUsed07 : INT ;
    NotUsed08 : INT ;
    NotUsed09 : INT ;
    NotUsed10 : INT ;
    NotUsed11 : INT ;
    NotUsed12 : INT ;
   END_STRUCT ;
   Hardware : STRUCT
    PLCBatteryFailure : BOOL ;
    NotUsed09 : BOOL ;
    NotUsed10 : BOOL ;
    NotUsed11 : BOOL ;
    NotUsed12 : BOOL ;
    NotUsed13 : BOOL ;
    NotUsed14 : BOOL ;
    NotUsed15 : BOOL ;
    VoltageOk : BOOL ;	//Control voltage ok
    EsGeneralOk : BOOL ;	//General emergency stop ok
    PowerOk : BOOL ;	//Power supply motor contactor panels ok
    FuseOk : BOOL ;	//Mini circuit breakers ok
    PlcOk : BOOL ;	//PLC ok
    FireOk : BOOL ;	//No fire alarms
    SmokeOk : BOOL ;	//No smoke alarms
    ExflapsOk : BOOL ;	//Explosion flaps ok
   END_STRUCT ;
   HardwareStop : STRUCT
    NotUsed08 : BOOL ;
    NotUsed09 : BOOL ;
    NotUsed10 : BOOL ;
    NotUsed11 : BOOL ;
    NotUsed12 : BOOL ;
    NotUsed13 : BOOL ;
    NotUsed14 : BOOL ;
    NotUsed15 : BOOL ;
    General : BOOL ;	//Stop from Hardware all circuits
    NotUsed01 : BOOL ;
    NotUsed02 : BOOL ;
    NotUsed03 : BOOL ;
    NotUsed04 : BOOL ;
    NotUsed05 : BOOL ;
    NotUsed06 : BOOL ;
    NotUsed07 : BOOL ;
   END_STRUCT ;
   GlobalFlags : STRUCT
    NotUsed08 : BOOL ;
    NotUsed09 : BOOL ;
    NotUsed10 : BOOL ;
    NotUsed11 : BOOL ;
    NotUsed12 : BOOL ;
    NotUsed13 : BOOL ;
    NotUsed14 : BOOL ;
    NotUsed15 : BOOL ;
    StaTest : BOOL ;	//Activates the test mode
    StaLOGOff : BOOL ;
    NotUsed02 : BOOL ;
    NotUsed03 : BOOL ;
    NotUsed04 : BOOL ;
    NotUsed05 : BOOL ;
    NotUsed06 : BOOL ;
    StaProtocolling : BOOL ;	//Activates the protocolling functionality of the elements
   END_STRUCT ;
   TestFunctions : STRUCT
    StaPLC1ComSimulation : BOOL ;
    StaPLC2ComSimulation : BOOL ;
    StaPLC3ComSimulation : BOOL ;
    StaPLC4ComSimulation : BOOL ;
    StaPLC5ComSimulation : BOOL ;
    NotUsed13 : BOOL ;
    NotUsed14 : BOOL ;
    NotUsed15 : BOOL ;
    StaIOManager : BOOL ;	//IO's simulated with the IO-Manager
    StaHardware : BOOL ;	//IO's connected to the real hardware
    StaCWASimulation : BOOL ;	//CWA-Simulator on
    StaIOSimuli : BOOL ;	//IO's simulated with the IOSimuli
    StaDPSimulation : BOOL ;
    StaWinAC : BOOL ;	//The PLC-Software runs on a WinAC-SoftPLC
    NotUsed06 : BOOL ;
    StaPCDirectInhouseTest : BOOL ;	//Direct control channel for inhouse test
   END_STRUCT ;
   PlantID : STRUCT
    Product : ARRAY  [1 .. 15 ] OF //i.e. MELE_SMU01_99
    CHAR ;
    PlcNr : INT  := 1;
    GCSRelease : INT  := 2;
   END_STRUCT ;
  END_STRUCT ;	
BEGIN
   PlantID.Product[1] := 'M';
   PlantID.Product[2] := 'E';
   PlantID.Product[3] := 'L';
   PlantID.Product[4] := 'E';
   PlantID.Product[5] := '_';
   PlantID.Product[6] := 'S';
   PlantID.Product[7] := 'M';
   PlantID.Product[8] := 'U';
   PlantID.Product[9] := '0';
   PlantID.Product[10] := '1';
   PlantID.Product[11] := '_';
   PlantID.Product[12] := '9';
   PlantID.Product[13] := '9';
   PlantID.Product[14] := ' ';
   PlantID.Product[15] := ' ';
   PlantID.PlcNr := 1;
   PlantID.GCSRelease := 2;
END_DATA_BLOCK

DATA_BLOCK "ASW_TimerSettings"	// DB 56
//COPYRIGHT:    (C) 2000 BY  BUHLER AG
//                           CH-9240 UZWIL  SWITZERLAND
//
//PRODUCT:     MELE_SMU01_99
//
//TITLE:        SYS: Default timer settings
//
//              SYS: Zeiteneinstellwerte
//
//
//--------------------------------------------------------------------------------
//
//IDENT:        AUTHOR:             DEPT:                              DATE:
//
//STD_DB056.1A  Ph. Engler          MU664                              05-Jan-2000
//              1st Release
//
//--------------------------------------------------------------------------------
//
//PURPOSE:  
//MANUAL : 
//CODE   :
//RESTRICTIONS:
//
//--------------------------------------------------------------------------------
//
//
//
//
//
//
//
AUTHOR : PE
FAMILY : USW
VERSION : 0.0
  STRUCT
   Notused : S5TIME ;
   Timer01 : S5TIME ;
   Timer02 : S5TIME ;
   Timer03 : S5TIME ;
   Timer04 : S5TIME ;
   Timer05 : S5TIME ;
   Timer06 : S5TIME ;
   Timer07 : S5TIME ;
   Timer08 : S5TIME ;
   Timer09 : S5TIME ;
   Timer10 : S5TIME  := S5T#10S;	//SYS: Delay after new- or restart
   Timer11 : S5TIME  := S5T#10S;	//SYS: Delay after hardware ok
   Timer12 : S5TIME ;
   Timer13 : S5TIME  := S5T#1S;	//SYS: Delay log entrys after fuse tripped
   Timer14 : S5TIME  := S5T#15S;	//SYS: Delay for section staOffline (section hangs in stEmptied)
   Timer15 : S5TIME  := S5T#2S;	//SYS: Offline time after a newstart
   Timer16 : S5TIME  := S5T#3M;	//SYS: Reset the "GCS7_Gr_InHeavyStartup" (M13.6) after this time
   Timer17 : S5TIME ;
   Timer18 : S5TIME ;
   Timer19 : S5TIME ;
   Timer20 : S5TIME  := S5T#1M;	//COM: PCCWatchdog
   Timer21 : S5TIME ;
   Timer22 : S5TIME ;
   Timer23 : S5TIME ;
   Timer24 : S5TIME ;
   Timer25 : S5TIME ;
   Timer26 : S5TIME ;
   Timer27 : S5TIME ;
   Timer28 : S5TIME ;
   Timer29 : S5TIME ;
   Timer30 : S5TIME ;
   Timer31 : S5TIME ;	//CWA01
   Timer32 : S5TIME ;	//CWA02
   Timer33 : S5TIME ;	//CWA03
   Timer34 : S5TIME ;	//CWA04
   Timer35 : S5TIME ;	//CWA05
   Timer36 : S5TIME ;	//CWA06
   Timer37 : S5TIME ;	//CWA07
   Timer38 : S5TIME ;	//CWA08
   Timer39 : S5TIME ;	//CWA09
   Timer40 : S5TIME ;	//CWA10
   Timer41 : S5TIME ;	//CWA11
   Timer42 : S5TIME ;	//CWA12
   Timer43 : S5TIME ;	//CWA13
   Timer44 : S5TIME ;	//CWA14
   Timer45 : S5TIME ;	//CWA15
   Timer46 : S5TIME ;	//CWA16
   Timer47 : S5TIME ;	//CWA17
   Timer48 : S5TIME ;	//CWA18
   Timer49 : S5TIME ;	//CWA19
   Timer50 : S5TIME ;	//CWA20
   Timer51 : S5TIME ;	//L01:
   Timer52 : S5TIME ;
   Timer53 : S5TIME ;
   Timer54 : S5TIME ;
   Timer55 : S5TIME ;
   Timer56 : S5TIME ;
   Timer57 : S5TIME ;
   Timer58 : S5TIME ;
   Timer59 : S5TIME ;
   Timer60 : S5TIME ;	//L01:
   Timer61 : S5TIME ;	//L02:
   Timer62 : S5TIME ;
   Timer63 : S5TIME ;
   Timer64 : S5TIME ;
   Timer65 : S5TIME ;
   Timer66 : S5TIME ;
   Timer67 : S5TIME ;
   Timer68 : S5TIME ;
   Timer69 : S5TIME ;
   Timer70 : S5TIME ;	//L02:
   Timer71 : S5TIME ;	//L03:
   Timer72 : S5TIME ;
   Timer73 : S5TIME ;
   Timer74 : S5TIME ;
   Timer75 : S5TIME ;
   Timer76 : S5TIME ;
   Timer77 : S5TIME ;
   Timer78 : S5TIME ;
   Timer79 : S5TIME ;
   Timer80 : S5TIME ;	//L03:
   Timer81 : S5TIME ;	//L04:
   Timer82 : S5TIME ;
   Timer83 : S5TIME ;
   Timer84 : S5TIME ;
   Timer85 : S5TIME ;
   Timer86 : S5TIME ;
   Timer87 : S5TIME ;
   Timer88 : S5TIME ;
   Timer89 : S5TIME ;
   Timer90 : S5TIME ;	//L04:
   Timer91 : S5TIME ;	//L05:
   Timer92 : S5TIME ;
   Timer93 : S5TIME ;
   Timer94 : S5TIME ;
   Timer95 : S5TIME ;
   Timer96 : S5TIME ;
   Timer97 : S5TIME ;
   Timer98 : S5TIME ;
   Timer99 : S5TIME ;
   Timer100 : S5TIME ;	//L05:
   Timer101 : S5TIME ;	//L06:
   Timer102 : S5TIME ;
   Timer103 : S5TIME ;
   Timer104 : S5TIME ;
   Timer105 : S5TIME ;
   Timer106 : S5TIME ;
   Timer107 : S5TIME ;
   Timer108 : S5TIME ;
   Timer109 : S5TIME ;
   Timer110 : S5TIME ;	//L06:
   Timer111 : S5TIME ;	//L07:
   Timer112 : S5TIME ;
   Timer113 : S5TIME ;
   Timer114 : S5TIME ;
   Timer115 : S5TIME ;
   Timer116 : S5TIME ;
   Timer117 : S5TIME ;
   Timer118 : S5TIME ;
   Timer119 : S5TIME ;
   Timer120 : S5TIME ;	//L07:
   Timer121 : S5TIME ;	//L08:
   Timer122 : S5TIME ;
   Timer123 : S5TIME ;
   Timer124 : S5TIME ;
   Timer125 : S5TIME ;
   Timer126 : S5TIME ;
   Timer127 : S5TIME ;
   Timer128 : S5TIME ;
   Timer129 : S5TIME ;
   Timer130 : S5TIME ;	//L08:
   Timer131 : S5TIME ;	//L09:
   Timer132 : S5TIME ;
   Timer133 : S5TIME ;
   Timer134 : S5TIME ;
   Timer135 : S5TIME ;
   Timer136 : S5TIME ;
   Timer137 : S5TIME ;
   Timer138 : S5TIME ;
   Timer139 : S5TIME ;
   Timer140 : S5TIME ;	//L09:
   Timer141 : S5TIME ;	//L10:
   Timer142 : S5TIME ;
   Timer143 : S5TIME ;
   Timer144 : S5TIME ;
   Timer145 : S5TIME ;
   Timer146 : S5TIME ;
   Timer147 : S5TIME ;
   Timer148 : S5TIME ;
   Timer149 : S5TIME ;
   Timer150 : S5TIME ;	//L10:
   Timer151 : S5TIME ;
   Timer152 : S5TIME ;
   Timer153 : S5TIME ;
   Timer154 : S5TIME ;
   Timer155 : S5TIME ;
   Timer156 : S5TIME ;
   Timer157 : S5TIME ;
   Timer158 : S5TIME ;
   Timer159 : S5TIME ;
   Timer160 : S5TIME ;
   Timer161 : S5TIME ;
   Timer162 : S5TIME ;
   Timer163 : S5TIME ;
   Timer164 : S5TIME ;
   Timer165 : S5TIME ;
   Timer166 : S5TIME ;
   Timer167 : S5TIME ;
   Timer168 : S5TIME ;
   Timer169 : S5TIME ;
   Timer170 : S5TIME ;
   Timer171 : S5TIME ;
   Timer172 : S5TIME ;
   Timer173 : S5TIME ;
   Timer174 : S5TIME ;
   Timer175 : S5TIME ;
   Timer176 : S5TIME ;
   Timer177 : S5TIME ;
   Timer178 : S5TIME ;
   Timer179 : S5TIME ;
   Timer180 : S5TIME ;
   Timer181 : S5TIME ;
   Timer182 : S5TIME ;
   Timer183 : S5TIME ;
   Timer184 : S5TIME ;
   Timer185 : S5TIME ;
   Timer186 : S5TIME ;
   Timer187 : S5TIME ;
   Timer188 : S5TIME ;
   Timer189 : S5TIME ;
   Timer190 : S5TIME ;
   Timer191 : S5TIME ;
   Timer192 : S5TIME ;
   Timer193 : S5TIME ;
   Timer194 : S5TIME ;
   Timer195 : S5TIME ;
   Timer196 : S5TIME ;
   Timer197 : S5TIME ;
   Timer198 : S5TIME ;
   Timer199 : S5TIME ;
   Timer200 : S5TIME ;
  END_STRUCT ;	
BEGIN
   Timer10 := S5T#10S;
   Timer11 := S5T#10S;
   Timer13 := S5T#1S;
   Timer14 := S5T#15S;
   Timer15 := S5T#2S;
   Timer16 := S5T#3M;
   Timer20 := S5T#1M;
END_DATA_BLOCK

